    IF _runOneStep THEN
        _runOneStep := FALSE;
        RETURN;
    END_IF
END_IF

IF SUPER^.Step(1008, TRUE, 'Step number 1008') THEN
    SUPER^.StepCompleteWhen((_runOneStep OR _runAllSteps) AND _finishStep);

    IF _runOneStep THEN
        _runOneStep := FALSE;
        RETURN;
    END_IF
END_IF

IF SUPER^.Step(1009, TRUE, 'Step number 1009') THEN
    SUPER^.StepCompleteWhen((_runOneStep OR _runAllSteps) AND _finishStep);

    IF _runOneStep THEN
        _runOneStep := FALSE;
        RETURN;
    END_IF
END_IF

IF SUPER^.Step(1010, TRUE, 'Step number 1010') THEN
    SUPER^.StepCompleteWhen((_runOneStep OR _runAllSteps) AND _finishStep);

    IF _runOneStep THEN
        _runOneStep := FALSE;
        RETURN;
    END_IF
END_IF

IF SUPER^.Step(1011, TRUE, 'Step number 1011') THEN
    SUPER^.StepCompleteWhen((_runOneStep OR _runAllSteps) AND _finishStep);

    IF _runOneStep THEN
        _runOneStep := FALSE;
        RETURN;
    END_IF
END_IF

IF SUPER^.Step(1012, TRUE, 'Step number 1012') THEN
    SUPER^.StepCompleteWhen((_runOneStep OR _runAllSteps) AND _finishStep);

    IF _runOneStep THEN
        _runOneStep := FALSE;
        RETURN;
    END_IF
END_IF

IF SUPER^.Step(1013, TRUE, 'Step number 1013') THEN
    SUPER^.StepCompleteWhen((_runOneStep OR _runAllSteps) AND _finishStep);

    IF _runOneStep THEN
        _runOneStep := FALSE;
        RETURN;
    END_IF
END_IF

IF SUPER^.Step(1014, TRUE, 'Step number 1014') THEN
    SUPER^.StepCompleteWhen((_runOneStep OR _runAllSteps) AND _finishStep);

    IF _runOneStep THEN
        _runOneStep := FALSE;
        RETURN;
    END_IF
END_IF

IF SUPER^.Step(1015, TRUE, 'Step number 1015') THEN
    SUPER^.StepCompleteWhen((_runOneStep OR _runAllSteps) AND _finishStep);

    IF _runOneStep THEN
        _runOneStep := FALSE;
        RETURN;
    END_IF
END_IF

IF SUPER^.Step(1016, TRUE, 'Step number 1016') THEN
    SUPER^.StepCompleteWhen((_runOneStep OR _runAllSteps) AND _finishStep);

    IF _runOneStep THEN
        _runOneStep := FALSE;
        RETURN;
    END_IF
END_IF

IF SUPER^.Step(1017, TRUE, 'Step number 1017') THEN
    SUPER^.StepCompleteWhen((_runOneStep OR _runAllSteps) AND _finishStep);

    IF _runOneStep THEN
        _runOneStep := FALSE;
        RETURN;
    END_IF
END_IF

IF SUPER^.Step(1018, TRUE, 'Step number 1018') THEN
    SUPER^.StepCompleteWhen((_runOneStep OR _runAllSteps) AND _finishStep);

    IF _runOneStep THEN
        _runOneStep := FALSE;
        RETURN;
    END_IF
END_IF

IF SUPER^.Step(1019, TRUE, 'Step number 1019') THEN
    SUPER^.StepCompleteWhen((_runOneStep OR _runAllSteps) AND _finishStep);

    IF _runOneStep THEN
        _runOneStep := FALSE;
        RETURN;
    END_IF
END_IF

IF SUPER^.Step(1020, TRUE, 'Step number 1020') THEN
    SUPER^.StepCompleteWhen((_runOneStep OR _runAllSteps) AND _finishStep);

    IF _runOneStep THEN
        _runOneStep := FALSE;
        RETURN;
    END_IF
END_IF

IF SUPER^.Step(1021, TRUE, 'Step number 1021') THEN
    SUPER^.StepCompleteWhen((_runOneStep OR _runAllSteps) AND _finishStep);

    IF _runOneStep THEN
        _runOneStep := FALSE;
        RETURN;
    END_IF
END_IF

IF SUPER^.Step(1022, TRUE, 'Step number 1022') THEN
    SUPER^.StepCompleteWhen((_runOneStep OR _runAllSteps) AND _finishStep);

    IF _runOneStep THEN
        _runOneStep := FALSE;
        RETURN;
    END_IF
END_IF

IF SUPER^.Step(1023, TRUE, 'Step number 1023') THEN
    SUPER^.StepCompleteWhen((_runOneStep OR _runAllSteps) AND _finishStep);

    IF _runOneStep THEN
        _runOneStep := FALSE;
        RETURN;
    END_IF
END_IF

//******************************************************************
IF SUPER^.Step(_stepId, _enabled, _stepDescription) THEN
    SUPER^.StepCompleteWhen((_runOneStep OR _runAllSteps) AND _finishStep);

    IF _runOneStep THEN
        _runOneStep := FALSE;
        RETURN;
    END_IF
END_IF
END_METHOD

METHOD PROTECTED OnSequenceCompleted
_onSequenceCompleteCount := _onSequenceCompleteCount + 1;
END_METHOD

METHOD PROTECTED OnSequencerError
VAR_INPUT
    inErrorId : eSequencerError;
END_VAR
CASE inErrorId OF
    eSequencerError.noError:
        _onSequencerErrorCount := _onSequencerErrorCount + 0;
    eSequencerError.NotUniqueStepId:
        _onSequencerErrorCount := _onSequencerErrorCount + 10;
    eSequencerError.StepIdHasBeenChanged:
        _onSequencerErrorCount := _onSequencerErrorCount + 20;
    eSequencerError.OrderOfTheStepHasBeenChanged:
        _onSequencerErrorCount := _onSequencerErrorCount + 40;
    eSequencerError.StepWithRequestedIdDoesNotExists:
        _onSequencerErrorCount := _onSequencerErrorCount + 50;
    eSequencerError.MultipleRequestStepMethodCall:
        _onSequencerErrorCount := _onSequencerErrorCount + 60;
    eSequencerError.StepIdTooLow:
        _onSequencerErrorCount := _onSequencerErrorCount + 70;
    eSequencerError.StepIdTooHigh:
        _onSequencerErrorCount := _onSequencerErrorCount + 80;
ELSE
    _onSequencerErrorCount := _onSequencerErrorCount + 0;
END_CASE
END_METHOD

METHOD PROTECTED OnStateChange
VAR_INPUT
    PreviousState : INT;
    NewState : INT;
END_VAR
THIS^._onStateChangeCount := THIS^._onStateChangeCount + 1;
_stateChangeFrom := PreviousState;
_stateChangeTo := NewState;

IF _callRestoreInOnStateChange THEN
    Restore();
END_IF
END_METHOD

METHOD PROTECTED OnStepCompleted
_onCompleteStepCount := _onCompleteStepCount + 1;
END_METHOD

PROPERTY INTERNAL RequestStepCycle : UINT
GET
RequestStepCycle := _requestStepCycle;
END_GET
SET
_requestStepCycle := RequestStepCycle;
END_SET
END_PROPERTY

METHOD INTERNAL SequencerClose
SUPER^._Close();
END_METHOD

METHOD INTERNAL SequencerHasError : BOOL
SequencerHasError := SUPER^._sequencerHasError;
END_METHOD

METHOD INTERNAL SequencerOpen
SUPER^._Open();
END_METHOD

METHOD INTERNAL SetChildState
VAR_INPUT
    inState : INT;
END_VAR
THIS^._myTcoState.ChangeState(inState);
END_METHOD

METHOD INTERNAL SetCurrentStep
VAR_INPUT
    inStepID : INT;
    inStepDescription : STRING(254);
END_VAR
THIS^._currentStep.ID := inStepID;
THIS^._currentStep.Description := inStepDescription;
END_METHOD

METHOD SetCurrentStepToErrorState : BOOL
_currentStep.Status := TcoCore.eStepStatus.Error;
SetCurrentStepToErrorState := _currentStep.Status = TcoCore.eStepStatus.Error;
END_METHOD

METHOD SetCyclicMode : BOOL
ModeController.Mode := eSequencerMode.CyclicMode;
SetCyclicMode := ModeController.Mode = eSequencerMode.CyclicMode;
END_METHOD

METHOD SetInvalidMode : BOOL
ModeController.Mode := eSequencerMode.Invalid;
SetInvalidMode := ModeController.Mode = eSequencerMode.Invalid;
END_METHOD

METHOD INTERNAL SetNumberOfSteps
VAR_INPUT
    inNumberOfSteps : UINT;
END_VAR
_stepCounter := inNumberOfSteps;
_numberOfStepsInSequence := inNumberOfSteps;
_previousNumberOfStepsInSequence := inNumberOfSteps;
END_METHOD

METHOD INTERNAL SetSequenceAsChecked
_stepIDUniquenessChecked := TRUE;
_StepIdUniquenessControlState := eStepIdUniquenessControlState.Done;
END_METHOD

METHOD INTERNAL SetSequenceAsNotChecked
_stepIDUniquenessChecked := FALSE;
_StepIdUniquenessControlState := eStepIdUniquenessControlState.NotYetStarted;
END_METHOD

METHOD SetStepMode : BOOL
ModeController.Mode := eSequencerMode.StepMode;
SetStepMode := ModeController.Mode = eSequencerMode.StepMode;
END_METHOD

METHOD INTERNAL SetTestParams
VAR_INPUT
    inRunOneStep : BOOL;
    inRunAllSteps : BOOL;
    inFinishStep : BOOL;
    inID : UINT;
    inEnabled : BOOL;
    inStepDescription : STRING(254);
END_VAR
THIS^._runOneStep := inRunOneStep;
THIS^._runAllSteps := inRunAllSteps;
THIS^._finishStep := inFinishStep;
THIS^._stepId := inID;
THIS^._enabled := inEnabled;
THIS^._stepDescription := inStepDescription;
END_METHOD

METHOD StepCount
VAR_INPUT
    inTotalStepNumber : UINT;
    inFinishStep : BOOL;
END_VAR
VAR
    i : INT;
    _lastStepId : INT;
END_VAR
FOR i := 0 TO inTotalStepNumber DO
    IF SUPER^.Step(i, TRUE, CONCAT('Step number ', INT_TO_STRING(i))) THEN
        SUPER^.StepCompleteWhen(inFinishStep);
    END_IF
END_FOR
END_METHOD

{attribute 'TcRpcEnable'}
METHOD INTERNAL UpdateCurrentStepDetails
_currentStepId := SUPER^._currentStep.ID;
_currentStepOrder := SUPER^._currentStep.Order;
_currentStepEnabled := SUPER^._currentStep.Enabled;
_currentStepDescription := SUPER^._currentStep.Description;
_currentStepStatus := SUPER^._currentStep.Status;
_currentStepDuration := SUPER^._currentStep.Duration;
END_METHOD

END_FUNCTION_BLOCK

// ---- Tests/TcoSequence/TcoSequenceNonAutoRestorableTest.TcPOU
FUNCTION_BLOCK TcoSequenceNonAutoRestorableTest EXTENDS TcoCore._internals_TcoContext
VAR
    _callMyPlcInstance : BOOL := FALSE;
    _sequencer : _TcoSequence(THIS^, eRestoreMode.None);
    _runPLCinstanceOnce : BOOL := FALSE;
    _runPLCinstanceCyclicaly : BOOL := FALSE;
    _stepID : INT := 32764;
    _enabled : BOOL;
    _stepDescription : STRING := 'Last step sequence message';
    _runOneStep : BOOL;
    _runAllSteps : BOOL;
    _finishStep : BOOL;
    _restore : BOOL;
    _cycleCount : INT;
    _restoreCycleCount : INT;
    _init : BOOL;
END_VAR

IF _callMyPlcInstance THEN
    IF NOT _init THEN
        ContextOpen();
        ContextClose();
        _init := THIS^._rtc.IsValid;
    END_IF

    IF _restore THEN
        ContextOpen();
        THIS^._sequencer.Restore();
        _restoreCycleCount := _restoreCycleCount + 1;
        _restore := FALSE;
        ContextClose();
        RETURN;
    END_IF

    IF _runPLCinstanceOnce AND NOT _runPLCinstanceCyclicaly THEN
        ContextOpen();
        THIS^.PLCinstanceRun(_stepID, _enabled, _stepDescription);
        _cycleCount := _cycleCount + 1;
        _runPLCinstanceOnce := FALSE;
        ContextClose();
    END_IF

    IF _runPLCinstanceCyclicaly AND NOT _runPLCinstanceOnce THEN
        ContextOpen();
        THIS^.PLCinstanceRun(_stepID, _enabled, _stepDescription);
        _cycleCount := _cycleCount + 1;
        ContextClose();
    END_IF
END_IF;

{attribute 'TcRpcEnable'}
METHOD ChildHasAutoRestoreEnabled : BOOL;
ChildHasAutoRestoreEnabled := _sequencer.ChildHasAutoRestoreEnabled();
END_METHOD

{attribute 'TcRpcEnable'}
METHOD ChildIsAutoRestorable : BOOL;
ChildIsAutoRestorable := _sequencer.ChildIsAutoRestorable();
END_METHOD

{attribute 'TcRpcEnable'}
METHOD CleanupPointers
_sequencer.CleanupPointers();
END_METHOD

{attribute 'TcRpcEnable'}
METHOD ClearNumberOfSteps
_sequencer.ClearNumberOfSteps();
END_METHOD

{attribute 'TcRpcEnable'}
METHOD PROTECTED ContextClose
SUPER^._Close();
END_METHOD

{attribute 'TcRpcEnable'}
METHOD ContextOpen
SUPER^._Open();
END_METHOD

{attribute 'TcRpcEnable'}
METHOD GetChildState : INT
GetChildState := _sequencer.GetChildState();
END_METHOD

{attribute 'TcRpcEnable'}
METHOD GetCurrentStepOrder : UINT
GetCurrentStepOrder := _sequencer._currentStep.Order;
END_METHOD

{attribute 'TcRpcEnable'}
METHOD GetNumberOfStepsInSequence : UINT
GetNumberOfStepsInSequence := _sequencer._numberOfStepsInSequence;
END_METHOD

{attribute 'TcRpcEnable'}
METHOD GetOrderOfTheCurrentlyEvaluatedStep : UINT
GetOrderOfTheCurrentlyEvaluatedStep := _sequencer._theOrderOfTheCurrentlyEvaluatedStep;
END_METHOD

{attribute 'TcRpcEnable'}
METHOD GetOrderOfTheCurrentlyExecutedStep : UINT
GetOrderOfTheCurrentlyExecutedStep := _sequencer._theOrderOfTheCurrentlyExecutedStep;
END_METHOD

{attribute 'TcRpcEnable'}
METHOD GetPreviousNumberOfStepsInSequence : UINT
GetPreviousNumberOfStepsInSequence := _sequencer._previousNumberOfStepsInSequence;
END_METHOD

{attribute 'TcRpcEnable'}
METHOD GetRequestStepCycle : UINT
GetRequestStepCycle := _sequencer.RequestStepCycle;
END_METHOD

{attribute 'TcRpcEnable'}
METHOD GetSequencerErrorId : INT
GetSequencerErrorId := _sequencer.GetSequencerErrorId();
END_METHOD

{attribute 'TcRpcEnable'}
METHOD GetTextOfTheMostImportantMessage : STRING(254)
GetTextOfTheMostImportantMessage := THIS^._sequencer.GetTextOfTheMostImportantMessage();
END_METHOD

{attribute 'TcRpcEnable'}
METHOD HasAutoRestoreEnabled : BOOL;
HasAutoRestoreEnabled := _sequencer.HasAutoRestoreEnabled();
END_METHOD

{attribute 'TcRpcEnable'}
METHOD IsAutoRestorable : BOOL;
IsAutoRestorable := _sequencer.IsAutoRestorable();
END_METHOD

{attribute 'TcRpcEnable'}
METHOD IsFirstStepEntry : BOOL
IsFirstStepEntry := THIS^._sequencer.IsFirstStepEntry();
END_METHOD

METHOD PROTECTED Main
END_METHOD

{attribute 'TcRpcEnable'}
METHOD PLCinstanceRun
VAR_INPUT
    inStepId : UINT;
    inEnabled : BOOL;
    inStepDescription : STRING(254);
END_VAR
THIS^._sequencer.SetTestParams(_runOneStep,
    _runAllSteps,
    _finishStep,
    inStepId,
    inEnabled,
    inStepDescription);

THIS^._sequencer._RunExecutionSubstitute();
END_METHOD

{attribute 'TcRpcEnable'}
METHOD RequestStep
VAR_INPUT
    inRequestedStepId : INT;
END_VAR
_sequencer._RequestStep(inRequestedStepId);
END_METHOD

{attribute 'TcRpcEnable'}
METHOD Restore
_sequencer.Restore();
END_METHOD

{attribute 'TcRpcEnable'}
METHOD SequenceComplete
_sequencer._SequenceComplete();
END_METHOD

{attribute 'TcRpcEnable'}
METHOD SequencerClose
THIS^._sequencer.SequencerClose();
END_METHOD

{attribute 'TcRpcEnable'}
METHOD SequencerHasError : BOOL
SequencerHasError := _sequencer.SequencerHasError();
END_METHOD

{attribute 'TcRpcEnable'}
METHOD SequencerOpen
THIS^._sequencer.SequencerOpen();
END_METHOD

{attribute 'TcRpcEnable'}
METHOD SetChildState
VAR_INPUT
    inState : INT;
END_VAR
_sequencer.SetChildState(inState);
END_METHOD

{attribute 'TcRpcEnable'}
METHOD SetCurrentStep
VAR_INPUT
    inStepID : INT;
    inStepDescription : STRING(254);
END_VAR
_sequencer.SetCurrentStep(inStepID := inStepID, inStepDescription := inStepDescription);
END_METHOD

{attribute 'TcRpcEnable'}
METHOD SetCurrentStepToErrorState : BOOL
SetCurrentStepToErrorState := _sequencer.SetCurrentStepToErrorState();
END_METHOD

{attribute 'TcRpcEnable'}
METHOD SetCyclicMode : BOOL
SetCyclicMode := _sequencer.SetCyclicMode();
END_METHOD

{attribute 'TcRpcEnable'}
METHOD SetInvalidMode : BOOL
SetInvalidMode := _sequencer.SetInvalidMode();
END_METHOD

{attribute 'TcRpcEnable'}
METHOD SetNumberOfSteps : UINT
VAR_INPUT
    inNumberOfSteps : UINT;
END_VAR
_sequencer.SetNumberOfSteps(inNumberOfSteps);
SetNumberOfSteps := _sequencer._numberOfStepsInSequence;
END_METHOD

{attribute 'TcRpcEnable'}
METHOD SetRequestStepCycle : UINT
VAR_INPUT
    Value : UINT;
END_VAR
_sequencer.RequestStepCycle := Value;
SetRequestStepCycle := _sequencer.RequestStepCycle;
END_METHOD

{attribute 'TcRpcEnable'}
METHOD SetSequenceAsChecked : BOOL
VAR_INPUT
END_VAR
_sequencer.SetSequenceAsChecked();
END_METHOD

{attribute 'TcRpcEnable'}
METHOD SetSequenceAsNotChecked : BOOL
VAR_INPUT
END_VAR
_sequencer.SetSequenceAsNotChecked();
END_METHOD

{attribute 'TcRpcEnable'}
METHOD SetStepMode : BOOL
SetStepMode := _sequencer.SetStepMode();
END_METHOD

{attribute 'TcRpcEnable'}
METHOD Step : BOOL
VAR_INPUT
    inStepId : INT;
    inEnabled : BOOL;
    inStepDescription : STRING(254);
END_VAR
Step := _sequencer._Step(inStepID := inStepId, inEnabled := inEnabled, inStepDescription := inStepDescription);
END_METHOD

{attribute 'TcRpcEnable'}
METHOD StepBackward
_sequencer._StepBackward();
END_METHOD

{attribute 'TcRpcEnable'}
METHOD StepCompleteWhen
VAR_INPUT
    inCondition : BOOL;
END_VAR
_sequencer._StepCompleteWhen(inCondition);
END_METHOD

{attribute 'TcRpcEnable'}
METHOD StepForward
_sequencer._StepForward();
END_METHOD

{attribute 'TcRpcEnable'}
METHOD StepIn
_sequencer._StepIn();
END_METHOD

{attribute 'TcRpcEnable'}
METHOD UpdateCurrentStepDetails
VAR_INPUT
END_VAR
_sequencer.UpdateCurrentStepDetails();
END_METHOD

END_FUNCTION_BLOCK

// ---- Tests/TcoMessenger/TcoMessengerContextTest.TcPOU
FUNCTION_BLOCK TcoMessengerContextTest EXTENDS TcoCore._internals_TcoContext
VAR
    _callMyPlcInstanceRtcUpdate : BOOL := FALSE;
    _callMyPlcInstanceRun : BOOL := FALSE;
    _nowLocal : DATE_AND_TIME;
    _nowUtc : DATE_AND_TIME;
    _rtcIsValid : BOOL := FALSE;
    _rtcIsSynchronized : BOOL := FALSE;
    {attribute addProperty Name "this is the name of messenger test"}
    _tcoMessangerTests : TcoMessengerTests(THIS^);
END_VAR

IF THIS^._callMyPlcInstanceRtcUpdate THEN
    THIS^._rtcUpdate();
    _nowLocal := THIS^.RealTimeClock.NowLocal();
    _nowUtc := THIS^.RealTimeClock.NowUTC();
    _rtcIsValid := THIS^.RealTimeClock.IsValid;
    _rtcIsSynchronized := THIS^.RealTimeClock.IsSynchronized;
END_IF

IF THIS^._callMyPlcInstanceRun THEN
    THIS^.Run();
END_IF

{attribute 'TcRpcEnable'}
METHOD INTERNAL ContextClose
SUPER^._Close();
END_METHOD

{attribute 'TcRpcEnable'}
METHOD INTERNAL ContextOpen
SUPER^._Open();
END_METHOD

METHOD PROTECTED Main
END_METHOD

{attribute 'TcRpcEnable'}
METHOD INTERNAL RtcIsValid : BOOL
RtcIsValid := THIS^.RealTimeClock.IsValid;
_rtcIsValid := THIS^.RealTimeClock.IsValid;
END_METHOD

END_FUNCTION_BLOCK

// ---- Tests/TcoMessenger/TcoMessengerTests.TcPOU
FUNCTION_BLOCK TcoMessengerTests EXTENDS TcoCore.TcoObject
VAR
    _category : TcoCore.eMessageCategory;
    _minLevel : TcoCore.eMessageCategory;
    _messageDigestMethod : TcoCore.eMessageDigestMethod;
    _messageLoggingMethod : TcoCore.eMessengerLogMethod;
END_VAR
VAR
    _BOOL : BOOL := TRUE;
    _BYTE : BYTE := 1;
    _WORD : WORD := 22;
    _DWORD : DWORD := 333;
    _LWORD : LWORD := 4444;
    _SINT : SINT := 12;
    _USINT : USINT := 13;
    _INT : INT := 14;
    _UINT : UINT := 55;
    _DINT : DINT := 66;
    _UDINT : UDINT := 77;
    _LINT : LINT := 88;
    _ULINT : ULINT := 99;
    _LTIME : LTIME := LTIME#551US615NS;
    _Real : REAL := 99.9;
    _LReal : LREAL := 88.8;
    _DateAndTime : DATE_AND_TIME := DT#2106-02-06-06:28:15;
    _Date : DATE := D#2106-02-06;
    _Time : TIME := T#71582M47S295MS;
    _WString : WSTRING := "W1";
    _TOD : TOD := TOD#23:59:59.999;
    _String : STRING := 'S1';
END_VAR

{attribute 'TcRpcEnable'}
METHOD AppendAnys_1 : BOOL
VAR_INPUT
END_VAR
_messenger.Build()
    .AppendAny(_BOOL)
    .AppendAny(_BYTE)
    .AppendAny(_WORD)
    .AppendAny(_DWORD)
    .AppendAny(_LWORD)
    .AppendAny(_SINT)
    .AppendAny(_USINT)
    .AppendAny(_INT)
    .AppendAny(_UINT)
    .AppendAny(_DINT)
    .AppendAny(_UDINT)
    .As().AsDebug();
END_METHOD

{attribute 'TcRpcEnable'}
METHOD AppendAnys_2 : BOOL
VAR_INPUT
END_VAR
_messenger.Build()
    .AppendAny(_LINT)
    .AppendAny(_ULINT)
    .AppendAny(_LTIME)
    .AppendAny(_Real)
    .AppendAny(_LReal)
    .AppendAny(_DateAndTime)
    .AppendAny(_Date)
    .AppendAny(_Time)
    .AppendAny(_WString)
    .AppendAny(_TOD)
    .AppendAny(_String)
    .As().AsDebug();
END_METHOD

{attribute 'TcRpcEnable'}
METHOD AsDebug : BOOL
VAR_INPUT
    TextMessage1 : STRING;
    TextMessage2 : STRING;
    Value : LREAL;
END_VAR
_messenger.Build().Append(TextMessage1).Append(TextMessage2).AppendAny(Value).As().AsDebug();
END_METHOD

{attribute 'TcRpcEnable'}
METHOD AsError : BOOL
VAR_INPUT
    TextMessage1 : STRING;
    TextMessage2 : STRING;
    Value : LREAL;
END_VAR
_messenger.Build().Append(TextMessage1).Append(TextMessage2).AppendAny(Value).As().AsError();
END_METHOD

{attribute 'TcRpcEnable'}
METHOD AsFatal : BOOL
VAR_INPUT
    TextMessage1 : STRING;
    TextMessage2 : STRING;
    Value : LREAL;
END_VAR
_messenger.Build().Append(TextMessage1).Append(TextMessage2).AppendAny(Value).As().AsFatal();
END_METHOD

{attribute 'TcRpcEnable'}
METHOD AsInfo : BOOL
VAR_INPUT
    TextMessage1 : STRING;
    TextMessage2 : STRING;
    Value : LREAL;
END_VAR
_messenger.Build().Append(TextMessage1).Append(TextMessage2).AppendAny(Value).As().AsInfo();
END_METHOD

{attribute 'TcRpcEnable'}
METHOD AsTrace : BOOL
VAR_INPUT
    TextMessage1 : STRING;
    TextMessage2 : STRING;
    Value : LREAL;
END_VAR
_messenger.Build().Append(TextMessage1).Append(TextMessage2).AppendAny(Value).As().AsTrace();
END_METHOD

{attribute 'TcRpcEnable'}
METHOD AsWarning : BOOL
VAR_INPUT
    TextMessage1 : STRING;
    TextMessage2 : STRING;
    Value : LREAL;
END_VAR
_messenger.Build().Append(TextMessage1).Append(TextMessage2).AppendAny(Value).As().AsWarning();
END_METHOD

{attribute 'TcRpcEnable'}
METHOD INTERNAL Catastrophic
VAR_INPUT
    Message : STRING(255);
END_VAR
_messenger.Catastrophic(Message);
END_METHOD

{attribute 'TcRpcEnable'}
METHOD INTERNAL Critical
VAR_INPUT
    Message : STRING(255);
END_VAR
_messenger.Critical(Message);
END_METHOD

{attribute 'TcRpcEnable'}
METHOD INTERNAL Debug
VAR_INPUT
    Message : STRING(255);
END_VAR
_messenger.Debug(Message);
END_METHOD

{attribute 'TcRpcEnable'}
METHOD INTERNAL Error
VAR_INPUT
    Message : STRING(255);
END_VAR
_messenger.Error(Message);
END_METHOD

{attribute 'TcRpcEnable'}
METHOD INTERNAL Info
VAR_INPUT
    Message : STRING(255);
END_VAR
_messenger.Info(Message);
END_METHOD

{attribute 'TcRpcEnable'}
METHOD INTERNAL Notify
VAR_INPUT
    Message : STRING(255);
END_VAR
_messenger.Notify(Message);
END_METHOD

{attribute 'TcRpcEnable'}
METHOD OnCondition : BOOL
VAR_INPUT
    inCondition : BOOL;
    message : STRING;
END_VAR
_messenger.OnCondition(inCondition).Post(message, _category);
END_METHOD

{attribute 'TcRpcEnable'}
METHOD Pin : BOOL
VAR_INPUT
    inCondition : BOOL;
    message : STRING;
END_VAR
IF (inCondition) THEN
    _messenger.Post(message, _category).Pin();
ELSE
    _messenger.Post(message, _category);
END_IF;
END_METHOD

{attribute 'TcRpcEnable'}
METHOD Pinned : BOOL
Pinned := _messenger.Pinned;
END_METHOD

{attribute 'TcRpcEnable'}
METHOD INTERNAL Post
VAR_INPUT
    Message : STRING(255);
END_VAR
_messenger.Post(Message, _category);
END_METHOD

{attribute 'TcRpcEnable'}
METHOD INTERNAL Programming
VAR_INPUT
    Message : STRING(255);
END_VAR
_messenger.Programming(Message);
END_METHOD

{attribute 'TcRpcEnable'}
METHOD INTERNAL Resume
Context.Environment.Messaging.Resume();
END_METHOD

{attribute 'TcRpcEnable'}
METHOD INTERNAL SetMessageDigestMethod
Context.Environment.Messaging.MessageDigestMethod := _messageDigestMethod;
END_METHOD

{attribute 'TcRpcEnable'}
METHOD INTERNAL SetMessageLoggingMethod
Context.Environment.Messaging.MessengerLoggingMethod := _messageLoggingMethod;
END_METHOD

{attribute 'TcRpcEnable'}
METHOD INTERNAL SetMinLevel
Context.Environment.Messaging.MinLevel := _minLevel;
END_METHOD

{attribute 'TcRpcEnable'}
METHOD INTERNAL Suspend
Context.Environment.Messaging.Suspend();
END_METHOD

{attribute 'TcRpcEnable'}
METHOD INTERNAL TimedOut
VAR_INPUT
    Message : STRING(255);
END_VAR
_messenger.Warning(Message);
END_METHOD

{attribute 'TcRpcEnable'}
METHOD INTERNAL Trace
VAR_INPUT
    Message : STRING(255);
END_VAR
_messenger.Trace(Message);
END_METHOD

{attribute 'TcRpcEnable'}
METHOD UnPin : BOOL
VAR_INPUT
    inCondition : BOOL;
    message : STRING;
END_VAR
_messenger.UnPin();
END_METHOD

{attribute 'TcRpcEnable'}
METHOD INTERNAL Warning
VAR_INPUT
    Message : STRING(255);
END_VAR
_messenger.Warning(Message);
END_METHOD

END_FUNCTION_BLOCK

// ---- Tests/TcoMessenger/TcoContextMessagingPerf.TcPOU
FUNCTION_BLOCK TcoContextMessagingPerf EXTENDS TcoContextTest
VAR
    _lot_of_messages : ARRAY[0.._messagesUpperBound] OF TcoCore.TcoMessenger(THIS^);
    _numberOfTestMessages : INT;
END_VAR
VAR CONSTANT
    _messagesUpperBound : INT := 10000;
END_VAR

METHOD PROTECTED Main
VAR
    index : INT;
END_VAR
IF (_numberOfTestMessages > _messagesUpperBound) THEN
    _numberOfTestMessages := _messagesUpperBound;
END_IF

FOR index := 0 TO _numberOfTestMessages DO
    THIS^._lot_of_messages[index].Info(INT_TO_STRING(index));
END_FOR
END_METHOD

END_FUNCTION_BLOCK

// ---- Tests/TcoComponent/TcoComponentTest.TcPOU
FUNCTION_BLOCK TcoComponentTest EXTENDS TcoCore._internals_TcoContext
VAR
    _callMyPlcInstance : BOOL := FALSE;
    _component : _TcoComponent(THIS^);
    _runPLCinstanceOnce : BOOL := FALSE;
    _runPLCinstanceCyclicaly : BOOL := FALSE;
    _restore : BOOL;
    _cycleCount : INT;
    _restoreCycleCount : INT;
    _init : BOOL;
END_VAR

IF _callMyPlcInstance THEN
    IF NOT _init THEN
        ContextOpen();
        ContextClose();
        _init := THIS^._rtc.IsValid;
    END_IF

    IF _restore THEN
        ContextOpen();
        THIS^._component.Restore();
        _restoreCycleCount := _restoreCycleCount + 1;
        _restore := FALSE;
        ContextClose();
        RETURN;
    END_IF

    IF _runPLCinstanceOnce AND NOT _runPLCinstanceCyclicaly THEN
        ContextOpen();
        THIS^.PLCinstanceRun();
        _cycleCount := _cycleCount + 1;
        _runPLCinstanceOnce := FALSE;
        ContextClose();
    END_IF

    IF _runPLCinstanceCyclicaly AND NOT _runPLCinstanceOnce THEN
        ContextOpen();
        THIS^.PLCinstanceRun();
        _cycleCount := _cycleCount + 1;
        ContextClose();
    END_IF
END_IF;

{attribute 'TcRpcEnable'}
METHOD INTERNAL ContextClose
SUPER^._Close();
END_METHOD

{attribute 'TcRpcEnable'}
METHOD INTERNAL ContextOpen
SUPER^._Open();
END_METHOD

{attribute 'TcRpcEnable'}
METHOD INTERNAL IsService : BOOL
IsService := THIS^._component.IsService;
END_METHOD

METHOD PROTECTED Main
END_METHOD

{attribute 'TcRpcEnable'}
METHOD INTERNAL PLCinstanceRun
THIS^._component();
END_METHOD

METHOD PROTECTED Restore
THIS^._component.Restore();
END_METHOD

{attribute 'TcRpcEnable'}
METHOD INTERNAL Service
THIS^._component.Service();
END_METHOD

{attribute 'TcRpcEnable'}
METHOD INTERNAL TriggerRestore
THIS^.Restore();
END_METHOD

END_FUNCTION_BLOCK

// ---- Tests/TcoComponent/_TcoComponent.TcPOU
FUNCTION_BLOCK _TcoComponent EXTENDS TcoCore.TcoComponent
VAR
    _task : TcoTaskTest(THIS^);
    _serviceModeCount : ULINT;
END_VAR

_task();

{attribute 'TcRpcEnable'}
METHOD INTERNAL CallBodyFromTest
_task();
END_METHOD

(*~
    <docu>
        <summary>
            Restores this instance to the Ready state. Can be called explicitly or from within one of the restore mechanisms.
        </summary>
    </docu>
~*)
METHOD Restore : ITcoRestorable
_task.Restore();
END_METHOD

METHOD PROTECTED ServiceMode
_serviceModeCount := _serviceModeCount + 1;
END_METHOD

END_FUNCTION_BLOCK

// ---- Tests/Utilities/StringBuilderTests.TcPOU
FUNCTION_BLOCK StringBuilderTests
VAR
    StringBuilder : TcoCore.StringBuilder();
    StringBuilderResult : STRING;
END_VAR

{attribute 'TcRpcEnable'}
METHOD Append
VAR_INPUT
    ToAppend : STRING;
END_VAR
StringBuilder.Append(ToAppend);
StringBuilderResult := StringBuilder._workString;
END_METHOD

{attribute 'TcRpcEnable'}
METHOD AppendAnyTest
StringBuilder.Clear();
// There was a strange compile-time error here... about function requiring exactly one input... could not get arround that... next time...
// 'AppendAny' is internal in the production code
//				     .AppendAny(_bool);
//					 .AppendAny(_real)
//					 .AppendAny(_lreal)
//					 .AppendAny(_dt)
//					 .AppendAny(_d)
//					 .AppendAny(_time)
//					 .AppendAny(_string)
//					 .AppendAny(_wstring)
//					 .AppendAny(_tod)
//					 .AppendAny(_int);
StringBuilderResult := StringBuilder._workString;
END_METHOD

{attribute 'TcRpcEnable'}
METHOD Clear
StringBuilder.Clear();
StringBuilderResult := StringBuilder._workString;
END_METHOD

{attribute 'TcRpcEnable'}
METHOD FluentApi : STRING
FluentApi :=
    StringBuilder.Clear().Append('1').Append('2').Append('3').Append('4').Clear().Append('1').Append('2').Append('3').Append('4').ToString();
END_METHOD

{attribute 'TcRpcEnable'}
METHOD ToString : STRING
ToString := StringBuilder.ToString();
StringBuilderResult := StringBuilder._workString;
END_METHOD

END_FUNCTION_BLOCK

// ---- Tests/TcoTask/PlcExecuted/TcoTaskTestContext.TcPOU
FUNCTION_BLOCK TcoTaskTestContext EXTENDS TcoCore._internals_TcoContext
VAR
    _sut : TcoCore.TcoTask(THIS^);
    _to_A : TcoTaskPlcTestObject(THIS^);
    _to_B : TcoTaskPlcTestObject(THIS^);
    _elapsedTimeETA : TIME;
    _elapsedTime : TIME;
    _runElapsedTimer : BOOL;
    _elapsedTimeTimer : Tc2_Standard.TON;
    _inBool : BOOL;
    _inUint : UINT;
    _inString : STRING;
    _retBool : BOOL;
    _retUint : UINT;
    _retString : STRING;
    _done : BOOL;
    _arranged : BOOL;
    _startCycles : ULINT;
    _endCycles : ULINT;
    _myIdentity : ULINT;
END_VAR

{attribute 'TcRpcEnable'}
METHOD _ClearPlcCycleCounter
ClearPlcCycleCounter();
END_METHOD

METHOD PROTECTED Main
_elapsedTimeTimer(IN := _runElapsedTimer, PT := _elapsedTimeETA);

CASE _testId OF
    {region "CallTasksBodiesOnly"}
    eTcoTaskTests.CallTasksBodiesOnly:
        _to_A();
        {endregion}
        {region "RestoreTasks"}
    eTcoTaskTests.RestoreTasks:
        _to_A._sut_A.Restore();
        _to_A._sut_B.Restore();
        _to_A();
        {endregion}
        {region "T300_TaskInvokeAndWaitForDone"}
    eTcoTaskTests.TaskInvokeAndWaitForDone:
        IF NOT _arranged THEN
            _to_A._sut_A.Restore();
            _to_A._sut_B.Restore();
            _to_A._sut_A.SetPreviousStateToReady();
            _to_A._sut_B.SetPreviousStateToReady();
            _arranged := TRUE;
        END_IF

        IF NOT _done THEN
            _to_A._sut_A.Invoke();
            _to_A._sut_B.Invoke();
            _to_A();
            _done := _to_A._sut_A.Done AND _to_A._sut_B.Done;
        END_IF

        IF _done THEN
            _to_A._sut_A.ReadOutState();
            _to_A._sut_B.ReadOutState();
            ProbeDoneWhen(_done);
        END_IF
        {endregion}
        {region "T301_TaskInvokeAfterDoneWithNoEmptyCycles"}
    eTcoTaskTests.TaskInvokeAfterDoneWithNoEmptyCycles:
        IF NOT _done THEN
            _to_A._sut_A.Invoke();
            _to_A._sut_B.Invoke();
            _to_A();
            _done := _to_A._sut_A.Done AND _to_A._sut_B.Done;
        END_IF

        IF _done THEN
            _to_A._sut_A.ReadOutState();
            _to_A._sut_B.ReadOutState();
            ProbeDoneWhen(_done);
        END_IF
        {endregion}
        {region "T302_TaskInvokeAfterDoneWithOneEmptyCycle"}
    eTcoTaskTests.TaskInvokeAfterDoneWithOneEmptyCycle:
        IF NOT _arranged THEN
            _arranged := TRUE;
            _plcCycleCounter := 0;
            RETURN;
        END_IF

        IF NOT _done THEN
            _to_A._sut_A.Invoke();
            _to_A._sut_B.Invoke();
            _to_A();
            _done := _to_A._sut_A.Done AND _to_A._sut_B.Done;
        END_IF

        IF _done THEN
            _to_A._sut_A.ReadOutState();
            _to_A._sut_B.ReadOutState();
            ProbeDoneWhen(_done);
        END_IF
        {endregion}
        {region "T303_TaskInvokeAfterDoneWithAbortCall"}
    eTcoTaskTests.TaskInvokeAfterDoneWithAbortCall:
        IF NOT _arranged THEN
            _to_A._sut_A.Abort();
            _to_A._sut_B.Abort();
            _arranged := TRUE;
        END_IF

        IF NOT _done THEN
            _to_A._sut_A.Invoke();
            _to_A._sut_B.Invoke();
            _to_A();
            _done := _to_A._sut_A.Done AND _to_A._sut_B.Done;
        END_IF

        IF _done THEN
            _to_A._sut_A.ReadOutState();
            _to_A._sut_B.ReadOutState();
            ProbeDoneWhen(_done);
        END_IF
        {endregion}
        {region "T304_TaskInvokeAfterDoneWithRestoreCall"}
    eTcoTaskTests.TaskInvokeAfterDoneWithRestoreCall:
        IF NOT _arranged THEN
            _to_A._sut_A.Restore();
            _to_A._sut_B.Restore();
            _arranged := TRUE;
        END_IF

        IF NOT _done THEN
            _to_A._sut_A.Invoke();
            _to_A._sut_B.Invoke();
            _to_A();
            _done := _to_A._sut_A.Done AND _to_A._sut_B.Done;
        END_IF

        IF _done THEN
            _to_A._sut_A.ReadOutState();
            _to_A._sut_B.ReadOutState();
            ProbeDoneWhen(_done);
        END_IF
        {endregion}
        {region "T305_TaskAbortDuringExecutionAndInvoke"}
    eTcoTaskTests.TaskAbortDuringExecutionAndInvoke:
        IF NOT _arranged THEN
            _arranged := TRUE;
            _plcCycleCounter := 0;
            _retBool := FALSE;
            RETURN;
        END_IF

        IF NOT _done THEN
            _to_A._sut_A.Invoke();
            _to_A._sut_B.Invoke();
            _to_A();

            IF _to_A._sut_A.Done AND NOT _retBool THEN
                _to_A._sut_A.Abort();
                _to_A._sut_B.Abort();
                _retBool := true;
            END_IF

            _done := _to_A._sut_A.Done AND _to_A._sut_B.Done;
        END_IF

        IF _done THEN
            _to_A._sut_A.ReadOutState();
            _to_A._sut_B.ReadOutState();
            ProbeDoneWhen(_done);
        END_IF
        {endregion}
        {region "T310_TaskError"}
    eTcoTaskTests.TaskError:
        IF NOT _arranged THEN
            IF _plcCycleCounter = 1 THEN
                _to_A.CounterValue_A := _inUint;
                RETURN;
            END_IF

            IF _plcCycleCounter = 2 THEN
                _to_A._sut_A.Invoke();
                RETURN;
            END_IF

            IF _plcCycleCounter > 2 AND _plcCycleCounter <= 5 THEN
                _to_A._sut_A();
                RETURN;
            END_IF

            IF _plcCycleCounter = 6 THEN
                _to_A._sut_A();
                _to_A._sut_A.ReadOutState();
                _arranged := TRUE;
                RETURN;
            END_IF
        END_IF

        IF NOT _done THEN
            IF _plcCycleCounter = 7 THEN
                _to_A.CounterValue_A := _to_A.CounterValue_A + 5;
                _to_A._sut_A();
                _to_A._sut_A.ReadOutState();
            END_IF

            IF _plcCycleCounter > 7 AND _plcCycleCounter <= 7 + _inUint THEN
                _to_A._sut_A();
                _to_A._sut_A.ReadOutState();
            END_IF

            _done := _plcCycleCounter >= 7 + _inUint;
            ProbeDoneWhen(_done);
        END_IF
        {endregion}
        {region "T311_TaskInvokeAfterErrorNoRestoreNoEmptyCycles"}
    eTcoTaskTests.TaskInvokeAfterErrorNoRestoreNoEmptyCycles:
        IF NOT _arranged THEN
            _to_A._sut_A.Invoke();
            _arranged := TRUE;
            RETURN;
        END_IF

        IF NOT _done THEN
            _to_A._sut_A();
            _to_A._sut_A.ReadOutState();
            ProbeDoneWhen(_plcCycleCounter >= 1 + _inUint);
        END_IF
        {endregion}
        {region "T312_TaskInvokeAfterErrorNoRestoreOneEmptyCycle"}
    eTcoTaskTests.TaskInvokeAfterErrorNoRestoreOneEmptyCycle:
        IF NOT _arranged THEN
            IF _plcCycleCounter = 1 THEN
                RETURN;
            END_IF

            IF _plcCycleCounter = 2 THEN
                _to_A._sut_A.Invoke();
                RETURN;
            END_IF
        END_IF

        IF NOT _done THEN
            _to_A._sut_A();
            _to_A._sut_A.ReadOutState();
            _done := _plcCycleCounter >= 2 + _inUint;
            ProbeDoneWhen(_done);
        END_IF
        {endregion}
        {region "T313_TaskInvokeAfterErrorWithRestore"}
    eTcoTaskTests.TaskInvokeAfterErrorWithRestore:
        _to_A._sut_A.Restore();
        _to_A._sut_A.Invoke();
        _to_A._sut_A();
        _to_A._sut_A.ReadOutState();
        _done := TRUE;
        ProbeDoneWhen(_done);
        {endregion}
        {region "T314_TaskAbortDuringExecution"}
    eTcoTaskTests.TaskAbortDuringExecution:
        IF _plcCycleCounter = 1 THEN
            _to_A._sut_A.Restore();
            RETURN;
        END_IF

        IF _plcCycleCounter = 2 THEN
            _to_A._sut_A.Invoke();
            _to_A._sut_A();
            _to_A._sut_A.ReadOutState();
            RETURN;
        END_IF

        IF _plcCycleCounter = 3 THEN
            _to_A._sut_A.Abort();
            _to_A._sut_A();
            _to_A._sut_A.ReadOutState();
            _done := TRUE;
            ProbeDoneWhen(_done);
        END_IF
        {endregion}
        {region "T315_TaskMessage"}
    eTcoTaskTests.TaskMessage:
        _to_A._sut_A.PostMessage(Message := _inString);
        _retString := _to_A._sut_A.GetMessage();
        _done := TRUE;
        ProbeDoneWhen(_done);
        {endregion}
        {region "T316_IdentitiesTest"}
    eTcoTaskTests.IdentitiesTest:
        _runElapsedTimer := TRUE;
        _elapsedTimeETA := UINT_TO_TIME(_inUint);
        _to_A._sut_A.ReadOutIdentities();
        _to_A.ReadOutIdentities();
        ReadOutCycleCounters();
        _done := _elapsedTimeTimer.Q;
        ProbeDoneWhen(_done);
        {endregion}
        {region "T317_CheckAutoRestoreProperties"}
    eTcoTaskTests.CheckAutoRestoreProperties:
        _to_A._tSt_A.ReadOutAutoRestoreProperties();
        _to_A._tSt_B.ReadOutAutoRestoreProperties();
        _to_A._tSt_A._tTt_A.ReadOutAutoRestoreProperties();
        _to_A._tSt_A._tTt_B.ReadOutAutoRestoreProperties();
        _to_A._tSt_B._tTt_A.ReadOutAutoRestoreProperties();
        _to_A._tSt_B._tTt_B.ReadOutAutoRestoreProperties();
        _done := TRUE;
        ProbeDoneWhen(_done);
        {endregion}
        {region "T318_AutoRestoreOnStateChange"}
    eTcoTaskTests.AutoRestoreOnStateChange:
        IF _plcCycleCounter = 1 THEN
            _to_A._tSt_A.ReadOutAutoRestoreProperties();
            _to_A._tSt_B.ReadOutAutoRestoreProperties();
            _to_A._tSt_A._tTt_A.ReadOutAutoRestoreProperties();
            _to_A._tSt_A._tTt_B.ReadOutAutoRestoreProperties();
            _to_A._tSt_B._tTt_A.ReadOutAutoRestoreProperties();
            _to_A._tSt_B._tTt_B.ReadOutAutoRestoreProperties();
            _to_A._tSt_A._tTt_A.ReadOutState();
            _to_A._tSt_B._tTt_B.ReadOutState();
        END_IF

        IF _plcCycleCounter = 2 THEN
            _to_A._tSt_A._tTt_A.Restore();
            _to_A._tSt_B._tTt_B.Restore();
            _to_A._tSt_A._tTt_A.ReadOutState();
            _to_A._tSt_B._tTt_B.ReadOutState();
        END_IF

        IF _plcCycleCounter = 3 THEN
            _to_A._tSt_A._tTt_A.Invoke();
            _to_A._tSt_B._tTt_B.Invoke();
            _to_A._tSt_A._tTt_A();
            _to_A._tSt_B._tTt_B();
            _to_A._tSt_A._tTt_A.ReadOutState();
            _to_A._tSt_B._tTt_B.ReadOutState();
        END_IF

        IF _plcCycleCounter = 4 THEN
            _to_A._tSt_A._tTt_A.Invoke();
            _to_A._tSt_A._tTt_A();
            _to_A._tSt_B._tTt_B();
            _to_A._tSt_A._tTt_A.ReadOutState();
            _to_A._tSt_B._tTt_B.ReadOutState();
        END_IF

        IF _plcCycleCounter = 5 THEN
            _to_A._tSt_A.ChangeState(_to_A._tSt_A._myState);
            _to_A._tSt_B.ChangeState(_to_A._tSt_B._myState);
            _to_A._tSt_A._tTt_A();
            _to_A._tSt_B._tTt_B();
            _to_A._tSt_A._tTt_A.ReadOutState();
            _to_A._tSt_B._tTt_B.ReadOutState();
        END_IF

        _done := _plcCycleCounter = 5;
        ProbeDoneWhen(_done);
        {endregion}
        {region "T320_InvokeDisabledTask"}
    eTcoTaskTests.InvokeDisabledTask:
        IF _plcCycleCounter = 1 THEN
            _to_A._sut_A.Restore();
            _to_A._sut_A.Disable();
            RETURN;
        END_IF

        IF NOT _done THEN
            _to_A._sut_A.Invoke();
            _to_A._sut_A();
            _to_A._sut_A.ReadOutState();
            _done := _plcCycleCounter >= 1 + _inUint;
            ProbeDoneWhen(_done);
        END_IF
        {endregion}
        {region "T321_DisableExecutingTask"}
    eTcoTaskTests.DisableExecutingTask:
        IF _plcCycleCounter = 1 THEN
            _to_A._sut_A.Enable();
            _to_A._sut_A.Invoke();
            _to_A._sut_A();
            _to_A._sut_A.ReadOutState();
            RETURN;
        END_IF

        IF _plcCycleCounter = 2 THEN
            _to_A._sut_A.Disable();
            _to_A._sut_A();
            _to_A._sut_A.ReadOutState();
            RETURN;
        END_IF

        IF _plcCycleCounter = 3 THEN
            _to_A._sut_A.Restore();
            _to_A._sut_A.Enable();
            _to_A._sut_A();
            _to_A._sut_A.ReadOutState();
            RETURN;
        END_IF

        IF _plcCycleCounter = 4 THEN
            _to_A._sut_A.Invoke();
            _to_A._sut_A();
            _to_A._sut_A.ReadOutState();
            RETURN;
        END_IF

        IF _plcCycleCounter = 5 THEN
            _to_A._sut_A.Restore();
            _to_A._sut_A();
            _to_A._sut_A.ReadOutState();
            _done := TRUE;
            ProbeDoneWhen(_done);
        END_IF
        {endregion}
        {region "T322_InvokeTaskThenDisable"}
    eTcoTaskTests.InvokeTaskThenDisable:
        _to_A._sut_A.Invoke();
        _to_A._sut_A.Disable();
        _to_A._sut_A();
        _to_A._sut_A.ReadOutState();
        _done := TRUE;
        ProbeDoneWhen(_done);
        {endregion}
        {region "T323_DisableTaskInErrorStateEnableAndTriggerAgain"}
    eTcoTaskTests.DisableTaskInErrorStateEnableAndTriggerAgain:
        IF _plcCycleCounter = 1 THEN
            _to_A._sut_A.Enable();
            _to_A._sut_A.Invoke();
            _to_A._sut_A();
            _to_A._sut_A.ReadOutState();
            RETURN;
        END_IF

        IF _plcCycleCounter = 2 THEN
            _to_A.CounterValue_A := _to_A.CounterValue_A + 5;
            _to_A._sut_A();
            _to_A._sut_A.ReadOutState();
            RETURN;
        END_IF

        IF _plcCycleCounter = 3 THEN
            _to_A._sut_A.Disable();
            _to_A._sut_A();
            _to_A._sut_A.ReadOutState();
            RETURN;
        END_IF

        IF _plcCycleCounter = 4 THEN
            _to_A._sut_A.Invoke();
            _to_A._sut_A();
            _to_A._sut_A.ReadOutState();
            RETURN;
        END_IF

        IF _plcCycleCounter = 5 THEN
            _to_A._sut_A.Restore();
            _to_A._sut_A.Invoke();
            _to_A._sut_A();
            _to_A._sut_A.ReadOutState();
            _done := TRUE;
            ProbeDoneWhen(_done);
        END_IF
        {endregion}
        {region "T330_ElapsedTypeMeasurement"}
    eTcoTaskTests.ElapsedTypeMeasurement:
        IF _plcCycleCounter = 1 THEN
            _to_A._sut_A.Restore();
            _to_A._sut_A.Enable();
            _to_A._sut_A.Invoke();
            RETURN;
        END_IF

        IF (_to_A._sut_A.Execute()) THEN
            _runElapsedTimer := TRUE;

            IF (_elapsedTimeTimer.Q) THEN
                _to_A._sut_A.DoneWhen(_elapsedTimeTimer.Q);
            END_IF;
        END_IF

        _done := _to_A._sut_A.Done;
        ProbeDoneWhen(_done);
        _elapsedTime := _to_A._sut_A.ElapsedTime;
        {endregion}
        {region "T340_TaskExecutingWithDoneAndErrorStatement"}
    eTcoTaskTests.TaskExecutingWithDoneAndErrorStatement:
        IF _plcCycleCounter = 1 THEN
            _to_A._sut_A.Restore();
            _to_A._sut_A.Enable();
            _to_A._sut_A.Invoke();
            _to_A._sut_A();
            _to_A._sut_A.ReadOutState();
            RETURN;
        END_IF

        _to_A._sut_A();
        _to_A._sut_A.DoneWhen(TRUE);
        _to_A._sut_A.ThrowWhen(TRUE);
        _to_A._sut_A.ReadOutState();
        _done := _to_A._sut_A.Done;
        ProbeDoneWhen(_done);
        {endregion}
        {region "T341_TaskExecutingWithErrorAndDoneStatement"}
    eTcoTaskTests.TaskExecutingWithErrorAndDoneStatement:
        IF _plcCycleCounter = 1 THEN
            _to_A._sut_A.Restore();
            _to_A._sut_A.Enable();
            _to_A._sut_A.Invoke();
            _to_A._sut_A();
            _to_A._sut_A.ReadOutState();
            RETURN;
        END_IF

        _to_A._sut_A();
        _to_A._sut_A.ThrowWhen(TRUE);
        _to_A._sut_A.DoneWhen(TRUE);
        _to_A._sut_A.ReadOutState();
        _done := _to_A._sut_A.Done;
        ProbeDoneWhen(_done);
        {endregion}
    eTcoTaskTests.TaskExecuteMethodNotCalled:
        _to_A._sut_A.Invoke().Done;
    eTcoTaskTests.TaskExecuteMethodCalled:
        _to_A._sut_A.Invoke().Done;
        _to_A._sut_A.Execute();
END_CASE
END_METHOD

METHOD INTERNAL ReadOutCycleCounters
_startCycles := THIS^.StartCycleCount;
_endCycles := THIS^.EndCycleCount;
_myIdentity := THIS^.Identity;
END_METHOD

END_FUNCTION_BLOCK

// ---- Tests/TcoTask/PlcExecuted/TcoTaskPlcTestObject.TcPOU
FUNCTION_BLOCK TcoTaskPlcTestObject EXTENDS TcoCore.TcoObject
VAR
    _myIdentity : ULINT;
    _myContextIdentity : ULINT;
    _myContextStartCount : ULINT;
    _myContextEndCount : ULINT;
    _myParentIdentity : ULINT;
    _sut_A : TcoTaskPlcTest(THIS^);
    _sut_B : TcoTaskPlcTest(THIS^);
    _tSt_A : TcoTaskPlcTestState(THIS^, eRestoreMode.AutoRestoreMembers);
    _tSt_B : TcoTaskPlcTestState(THIS^, eRestoreMode.None);
END_VAR

_sut_A();
_sut_B();

PROPERTY CounterValue_A : ULINT
GET
CounterValue_A := _sut_A.CounterValue;
END_GET
SET
_sut_A.CounterValue := CounterValue_A;
END_SET
END_PROPERTY

PROPERTY CounterValue_B : ULINT
GET
CounterValue_B := _sut_B.CounterValue;
END_GET
SET
_sut_B.CounterValue := CounterValue_B;
END_SET
END_PROPERTY

{attribute 'TcRpcEnable'}
METHOD INTERNAL ReadOutIdentities
_myIdentity := THIS^.Identity;
_myContextIdentity := THIS^.Context.Identity;
_myContextStartCount := THIS^.Context.StartCycleCount;
_myContextEndCount := THIS^.Context.EndCycleCount;
_myParentIdentity := THIS^.Parent.Identity;
END_METHOD

END_FUNCTION_BLOCK

// ---- Tests/TcoTask/PlcExecuted/TcoTaskPlcTest.TcPOU
FUNCTION_BLOCK TcoTaskPlcTest EXTENDS TcoCore.TcoTask
VAR
    _isBusy : BOOL;
    _isError : BOOL;
    _isDone : BOOL;
    _isReady : BOOL;
    _isInvokeRequestTrue : BOOL;
    _counterSetValue : ULINT;
    _counterValue : ULINT;
    _invokeCounter : ULINT;
    _executeCounter : ULINT;
    _doneCounter : ULINT;
    _invokeRisingEdgeCounter : ULINT;
    _executeRisingEdgeCounter : ULINT;
    _doneRisingEdgeCounter : ULINT;
    _previousState : eTaskState;
    _counterValuePV : ULINT;
    _myIdentity : ULINT;
    _myContextIdentity : ULINT;
    _myContextStartCount : ULINT;
    _myContextEndCount : ULINT;
    _myParentIdentity : ULINT;
    _autoRestoreByMyParentEnabled : BOOL;
    _onErrorCounter : ULINT;
    _whileErrorCounter : ULINT;
    _onStartCounter : ULINT;
END_VAR

IF (THIS^._taskState = eTaskState.Requested) THEN
    _invokeCounter := _invokeCounter + 1;
END_IF;

IF (THIS^._taskState = eTaskState.Requested AND _PreviousState <> eTaskState.Requested) THEN
    _counterValue := _counterSetValue;
    _counterValuePV := _counterValue;
    _invokeRisingEdgeCounter := _invokeRisingEdgeCounter + 1;
END_IF

IF (THIS^._taskState = eTaskState.Busy AND _previousState <> eTaskState.Busy) THEN
    _executeRisingEdgeCounter := _executeRisingEdgeCounter + 1;
END_IF

_previousState := THIS^._taskState;

IF (Execute()) THEN
    _executeCounter := _executeCounter + 1;
    _counterValue := _counterValue - 1;
    DoneWhen(_counterValue <= 0);
    ThrowWhen(ABS(_counterValuePV - _counterValue) > 1);
    _CounterValuePV := _counterValue;
END_IF

IF (THIS^._taskState = eTaskState.Done) THEN
    _doneCounter := _doneCounter + 1;
END_IF;

IF (THIS^._taskState = eTaskState.Done AND _previousState <> eTaskState.Done) THEN
    _doneRisingEdgeCounter := _doneRisingEdgeCounter + 1;
END_IF

PROPERTY CounterValue : ULINT
GET
CounterValue := _counterValue;
END_GET
SET
_counterValue := CounterValue;
END_SET
END_PROPERTY

METHOD INTERNAL Disable
THIS^.Enabled := FALSE;
END_METHOD

METHOD INTERNAL Enable
THIS^.Enabled := TRUE;
END_METHOD

METHOD INTERNAL GetMessage : STRING
GetMessage := SUPER^._messenger._mime.Text;
END_METHOD

METHOD PROTECTED OnError
_onErrorCounter := _onErrorCounter + 1;
END_METHOD

METHOD PROTECTED OnStart
_onStartCounter := _onStartCounter + 1;
END_METHOD

METHOD INTERNAL PostMessage
VAR_INPUT
    Message : STRING;
END_VAR
THIS^.Messenger.Post(Message, eMessageCategory.Error);
END_METHOD

{attribute 'TcRpcEnable'}
METHOD INTERNAL ReadOutAutoRestoreProperties
_autoRestoreByMyParentEnabled := THIS^.AutoRestorable;
END_METHOD

{attribute 'TcRpcEnable'}
METHOD INTERNAL ReadOutIdentities
_myIdentity := THIS^.Identity;
_myContextIdentity := THIS^.Context.Identity;
_myContextStartCount := THIS^.Context.StartCycleCount;
_myContextEndCount := THIS^.Context.EndCycleCount;
_myParentIdentity := THIS^.Parent.Identity;
END_METHOD

{attribute 'TcRpcEnable'}
METHOD INTERNAL ReadOutState
_isBusy := THIS^.Busy;
_isError := THIS^.Error;
_isDone := THIS^.Done;
_isReady := THIS^.Ready;
_isInvokeRequestTrue := THIS^._invokeRequest;
END_METHOD

{attribute 'TcRpcEnable'}
METHOD INTERNAL SetInvokeRequest
THIS^._invokeRequest := TRUE;
END_METHOD

{attribute 'TcRpcEnable'}
METHOD INTERNAL SetPreviousStateToReady
THIS^._previousState := eTaskState.Ready;
END_METHOD

(*~
    <docu>
        <summary>
            Executes until task is in ```Error``` state .
        </summary>
    </docu>
~*)
METHOD PROTECTED WhileError
_whileErrorCounter := _whileErrorCounter + 1;
END_METHOD

END_FUNCTION_BLOCK

// ---- Tests/TcoTask/PlcExecuted/TcoTaskPlcTestState.TcPOU
FUNCTION_BLOCK TcoTaskPlcTestState EXTENDS TcoState
VAR
    _myIdentity : ULINT;
    _myContextIdentity : ULINT;
    _myContextStartCount : ULINT;
    _myContextEndCount : ULINT;
    _myParentIdentity : ULINT;
    _myState : INT;
    _tTt_A : TcoTaskPlcTest(THIS^);
    _tTt_B : TcoTaskPlcTest(THIS^);
    _onStateChangeCounter : INT;
    _autoRestoreToMyChildsEnabled : BOOL;
    _autoRestoreByMyParentEnabled : BOOL;
END_VAR

METHOD PROTECTED OnStateChange
VAR_INPUT
    PreviousState : INT;
    NewState : INT;
END_VAR
VAR
    message : STRING;
END_VAR
_onStateChangeCounter := _onStateChangeCounter + 1;
message := CONCAT('My state has been change from ', INT_TO_STRING(PreviousState));
message := CONCAT(message, ' to the new state ');
message := CONCAT(message, INT_TO_STRING(NewState));
message := CONCAT(message, '.');
THIS^.Messenger.Post(message, eMessageCategory.Debug);
SUPER^.OnStateChange(PreviousState, NewState);
END_METHOD

{attribute 'TcRpcEnable'}
METHOD INTERNAL ReadOutAutoRestoreProperties
_autoRestoreToMyChildsEnabled := THIS^.IsAutoRestoreEnabled;
_autoRestoreByMyParentEnabled := THIS^.AutoRestorable;
END_METHOD

{attribute 'TcRpcEnable'}
METHOD INTERNAL ReadOutIdentities
_myIdentity := THIS^.Identity;
_myContextIdentity := THIS^.Context.Identity;
_myParentIdentity := THIS^.Parent.Identity;
_myContextStartCount := THIS^.Context.StartCycleCount;
_myContextEndCount := THIS^.Context.EndCycleCount;
END_METHOD

{attribute 'TcRpcEnable'}
METHOD INTERNAL ReadOutState
_myState := THIS^.State;
THIS^._tTt_A.ReadOutState();
THIS^._tTt_B.ReadOutState();
END_METHOD

{attribute 'TcRpcEnable'}
METHOD INTERNAL TriggerChangeState
VAR_INPUT
    NewState : INT;
END_VAR
THIS^.ChangeState(NewState);
END_METHOD

{attribute 'TcRpcEnable'}
METHOD INTERNAL TriggerChangeStateWithObjectRestore
VAR_INPUT
    NewState : INT;
END_VAR
THIS^.ChangeState(NewState).RestoreObject(THIS^._tTt_A).RestoreObject(THIS^._tTt_B);
END_METHOD

{attribute 'TcRpcEnable'}
METHOD INTERNAL TriggerRestore
THIS^.Restore();
END_METHOD

{attribute 'TcRpcEnable'}
METHOD INTERNAL TriggerTaskInvoke
THIS^._tTt_A.Invoke();
THIS^._tTt_B.Invoke();
END_METHOD

END_FUNCTION_BLOCK

// ---- Tests/TcoToggleTask/TcoToggleTaskTestContext.TcPOU
FUNCTION_BLOCK TcoToggleTaskTestContext EXTENDS TcoCore._internals_TcoContext
VAR
    _sut : TcoToggleTaskTests(THIS^, TRUE);
    _bool : BOOL;
    _string : STRING;
    _done : BOOL;
END_VAR

METHOD PROTECTED Main
CASE _testId OF
    eTcoToggleTaskTests.Reinit:
        _sut.FB_init(TRUE,
            FALSE,
            THIS^,
            _bool);

        _done := TRUE;
    eTcoToggleTaskTests.CleanUp:
        IF NOT _done THEN
            _sut._messenger.Clear();
            _done := TRUE;
        END_IF
    eTcoToggleTaskTests.Message:
        IF NOT _done THEN
            _sut.Messenger.Error(_string);
            _done := TRUE;
        END_IF
    eTcoToggleTaskTests.TriggerToggleWhileRunNotCalled:
        IF NOT _done THEN
            _sut._messenger.Clear();
            _sut.Toggle();
            _done := TRUE;
        END_IF
    eTcoToggleTaskTests.TriggerToggleWhileDisabled:
        IF NOT _done THEN
            _sut.Run();
            _sut._messenger.Clear();
            _sut.Enabled := FALSE;
            _sut.Toggle();
            _done := TRUE;
        END_IF
    eTcoToggleTaskTests.TriggerToggleWhileEnabled:
        IF NOT _done THEN
            _sut.Run();
            _sut._messenger.Clear();
            _sut.Enabled := TRUE;
            _sut.Toggle();
            _done := TRUE;
        END_IF
    eTcoToggleTaskTests.TriggerOnWhileRunNotCalled:
        IF NOT _done THEN
            _sut._messenger.Clear();
            _sut.On();
            _done := TRUE;
        END_IF
    eTcoToggleTaskTests.TriggerOnWhileDisabled:
        IF NOT _done THEN
            _sut.Run();
            _sut._messenger.Clear();
            _sut.Enabled := FALSE;
            _sut.On();
            _done := TRUE;
        END_IF
    eTcoToggleTaskTests.TriggerOnWhileEnabled:
        IF NOT _done THEN
            _sut.Run();
            _sut._messenger.Clear();
            _sut.Enabled := TRUE;
            _sut.On();
            _done := TRUE;
        END_IF
    eTcoToggleTaskTests.TriggerOffWhileRunNotCalled:
        IF NOT _done THEN
            _sut._messenger.Clear();
            _sut.Toggle();
            _done := TRUE;
        END_IF
    eTcoToggleTaskTests.TriggerOffWhileDisabled:
        IF NOT _done THEN
            _sut.Run();
            _sut._messenger.Clear();
            _sut.Enabled := FALSE;
            _sut.Off();
            _done := TRUE;
        END_IF
    eTcoToggleTaskTests.TriggerOffWhileEnabled:
        IF NOT _done THEN
            _sut.Run();
            _sut._messenger.Clear();
            _sut.Enabled := TRUE;
            _sut.Off();
            _done := TRUE;
        END_IF
END_CASE
END_METHOD

END_FUNCTION_BLOCK

// ---- Tests/TcoToggleTask/TcoToggleTaskTests.TcPOU
FUNCTION_BLOCK TcoToggleTaskTests EXTENDS TcoCore.TcoToggleTask
VAR
    _isOn : BOOL;
    _isOff : BOOL;
    _isEnabled : BOOL;
    _isToggleRequestTrue : BOOL;
    _counterValue : ULINT;
    _counterValuePV : ULINT;
    _toggleCounter : ULINT;
    _runCounter : ULINT;
    _onFtrigCounter : ULINT;
    _onRtrigCounter : ULINT;
    _onCounter : ULINT;
    _offCounter : ULINT;
    _onStateChangeCounter : ULINT;
    _taskOnCounter : ULINT;
    _taskOffCounter : ULINT;
    _stateChangedCounter : ULINT;
    _previousState : BOOL;
    _myIdentity : ULINT;
    _myContextIdentity : ULINT;
    _myContextStartCount : ULINT;
    _myContextEndCount : ULINT;
    _myParentIdentity : ULINT;
END_VAR

ExecutionBody();

METHOD INTERNAL Disable
THIS^.Enabled := FALSE;
END_METHOD

METHOD INTERNAL Enable
THIS^.Enabled := TRUE;
END_METHOD

{attribute 'TcRpcEnable'}
METHOD INTERNAL ExecutionBody
Run();
_runCounter := _runCounter + 1;

IF _previousState <> THIS^.State THEN
    _stateChangedCounter := _stateChangedCounter + 1;
END_IF;

_previousState := THIS^.State;
END_METHOD

{attribute 'TcRpcEnable'}
METHOD INTERNAL GetMessage : STRING
GetMessage := SUPER^._messenger._mime.Text;
END_METHOD

METHOD PROTECTED Main
VAR
END_VAR
END_METHOD

(*~
    <docu>
        <summary>
            Executes when toggle task changes its state from '''TRUE''' to '''FALSE'''.
        </summary>
    </docu>
~*)
METHOD PROTECTED OnFtrig
_onFtrigCounter := _onFtrigCounter + 1;
END_METHOD

(*~
    <docu>
        <summary>
            Executes when toggle task changes its state from '''FALSE''' to '''TRUE'''.
        </summary>
    </docu>
~*)
METHOD PROTECTED OnRtrig
_onRtrigCounter := _onRtrigCounter + 1;
END_METHOD

(*~
    <docu>
        <summary>
            Executes when toggle task changes its state .
        </summary>
    </docu>
~*)
METHOD PROTECTED OnStateChange
_onStateChangeCounter := _onStateChangeCounter + 1;
END_METHOD

{attribute 'TcRpcEnable'}
METHOD INTERNAL PostMessage
VAR_INPUT
    Message : STRING;
END_VAR
THIS^.Messenger.Post(Message, eMessageCategory.Error);
END_METHOD

{attribute 'TcRpcEnable'}
METHOD INTERNAL ReadOutIdentities
_myIdentity := THIS^.Identity;
_myContextIdentity := THIS^.Context.Identity;
_myContextStartCount := THIS^.Context.StartCycleCount;
_myContextEndCount := THIS^.Context.EndCycleCount;
_myParentIdentity := THIS^.Parent.Identity;
END_METHOD

{attribute 'TcRpcEnable'}
METHOD INTERNAL ReadOutState
_isOn := THIS^.IsOn;
_isOff := THIS^.IsOff;
_isEnabled := THIS^.Enabled;
_isToggleRequestTrue := THIS^._toggleRequest;
END_METHOD

{attribute 'TcRpcEnable'}
METHOD INTERNAL SetPreviousState
VAR_INPUT
    inValue : BOOL;
END_VAR
THIS^._previousState := inValue;
END_METHOD

{attribute 'TcRpcEnable'}
METHOD INTERNAL SetState
VAR_INPUT
    inState : BOOL;
END_VAR
THIS^._state := inState;
END_METHOD

{attribute 'TcRpcEnable'}
METHOD INTERNAL SetToggleRequest
THIS^._toggleRequest := TRUE;
END_METHOD

(*~
    <docu>
        <summary>
            Executes when toggle task is in ```Off``` state .
        </summary>
    </docu>
~*)
METHOD PROTECTED TaskOff
_taskOffCounter := _taskOffCounter + 1;
_counterValue := _counterValue - 1;
_CounterValuePV := _counterValue;
END_METHOD

(*~
    <docu>
        <summary>
            Executes when toggle task is in  ```On``` state .
        </summary>
    </docu>
~*)
METHOD PROTECTED TaskOn
_taskOnCounter := _taskOnCounter + 1;
_counterValue := _counterValue + 1;
_CounterValuePV := _counterValue;
END_METHOD

{attribute 'TcRpcEnable'}
METHOD INTERNAL TriggerOff
THIS^.Off();
_offCounter := _offCounter + 1;
END_METHOD

{attribute 'TcRpcEnable'}
METHOD INTERNAL TriggerOn
THIS^.On();
_onCounter := _onCounter + 1;
END_METHOD

{attribute 'TcRpcEnable'}
METHOD INTERNAL TriggerToggle
THIS^.Toggle();
_toggleCounter := _toggleCounter + 1;
END_METHOD

END_FUNCTION_BLOCK

// ---- Tests/TcoComponent/PlcExecuted/TcoComponentTestContext.TcPOU
FUNCTION_BLOCK TcoComponentTestContext EXTENDS TcoCore._internals_TcoContext
VAR
    _sut : TestComponent(THIS^);
    {attribute addProperty Name "--Some IO signal"}
    _signal : BOOL;
END_VAR

METHOD PROTECTED Main
CASE _testId OF
    eTcoComponentTests.GetSignalInfo:
        _sut(_signal := _signal);
END_CASE
END_METHOD

END_FUNCTION_BLOCK

// ---- Tests/TcoComponent/PlcExecuted/TestComponent.TcPOU
FUNCTION_BLOCK TestComponent EXTENDS TcoCore.TcoComponent
VAR_IN_OUT
    _signal : BOOL;
END_VAR
VAR
    _signalInfo : TcoCore.TcoSignalInfo;
END_VAR

_signalInfo.GetSignalInfo(SIZEOF(_signal), ADR(_signal));

(*~
    <docu>
        <summary>
            Restores this instance to the Ready state. Can be called explicitly or from within one of the restore mechanisms.
        </summary>
    </docu>
~*)
METHOD Restore : ITcoRestorable
END_METHOD

(*~
    <docu>
        <summary>
            Custom service (manual, maintenance) logic.
            This method must be implemented in derived class.
        </summary>
    </docu>
~*)
METHOD PROTECTED ServiceMode
END_METHOD

END_FUNCTION_BLOCK

// ---- Tests/TcoRemoteTask/PlcExecuted/TcoRemoteTaskTestContext.TcPOU
FUNCTION_BLOCK TcoRemoteTaskTestContext EXTENDS TcoCore._internals_TcoContext
VAR
    _sut : TcoRemoteTaskTest(THIS^);
    _invokeInitializedCSharpMethodDone : BOOL;
    _invokeNotInitializedCSharpMethodDone : BOOL;
    _exceptionInMethodWillResultInExceptionDone : BOOL;
    _sharedVariable : INT;
END_VAR

METHOD PROTECTED Main
CASE _testId OF
    0:
        _invokeInitializedCSharpMethodDone := FALSE;
        _invokeNotInitializedCSharpMethodDone := FALSE;
        _exceptionInMethodWillResultInExceptionDone := FALSE;
    eTcoRemoteTaskTests.RestoreTasks:
        _sut._invokeInitializedCSharpMethod.Restore();
        _sut._invokeNotInitializedCSharpMethod.Restore();
        _sut._exceptionInMethodWillResultInException.Restore();
    eTcoRemoteTaskTests.InvokeInitializedCSharpMethod:
        _invokeInitializedCSharpMethodDone := _sut._invokeInitializedCSharpMethod.Invoke().Done;
    eTcoRemoteTaskTests.InvokeNotInitializedCSharpMethod:
        _invokeNotInitializedCSharpMethodDone := _sut._invokeNotInitializedCSharpMethod.Invoke().Error;
    eTcoRemoteTaskTests.ExceptionInMethodWillResultInException:
        _exceptionInMethodWillResultInExceptionDone := _sut._exceptionInMethodWillResultInException.Invoke().Error;
END_CASE

_sut();
END_METHOD

END_FUNCTION_BLOCK

// ---- Tests/TcoRemoteTask/PlcExecuted/TcoRemoteTaskTest.TcPOU
FUNCTION_BLOCK TcoRemoteTaskTest EXTENDS TcoCore.TcoObject
VAR
    _invokeInitializedCSharpMethod : TcoCore.TcoRemoteTask(THIS^);
    _invokeNotInitializedCSharpMethod : TcoCore.TcoRemoteTask(THIS^);
    _exceptionInMethodWillResultInException : TcoCore.TcoRemoteTask(THIS^);
END_VAR

_invokeInitializedCSharpMethod();
_invokeNotInitializedCSharpMethod();
_exceptionInMethodWillResultInException();

END_FUNCTION_BLOCK

// ---- Tests/TcoSequencer/PlcExecuted/TcoSequencerTestContext.TcPOU
FUNCTION_BLOCK TcoSequencerTestContext EXTENDS TcoCore._internals_TcoContext
VAR
    _sut_A : TcoSequencerTestType(THIS^, eRestoreMode.AutoRestoreMembers);
    _sut_N : TcoSequencerTestType(THIS^, eRestoreMode.None);
    _elapsedTimeETA : TIME;
    _elapsedTime : TIME;
    _runElapsedTimer : BOOL;
    _elapsedTimeTimer : Tc2_Standard.TON;
    _runOneStep : BOOL;
    _runAllSteps : BOOL;
    _finishStep : BOOL;
    _stepId : INT;
    _enabled : BOOL;
    _stepDescription : STRING(254);
    _currentStepId : INT;
    _currentStepDescription : STRING(254);
    _totalStepNumber : UINT;
    _reqStep : INT;
    _reqStepNotExists : INT;
    _done : BOOL;
    _arranged : BOOL;
    _startCycles : ULINT;
    _endCycles : ULINT;
    _myIdentity : ULINT;
    _initReqStepCycle : UINT;
    _cycles : UINT;
    _cyclicCycles : UINT;
    _stepInEvents : UINT;
END_VAR

{attribute 'TcRpcEnable'}
METHOD _ClearPlcCycleCounter
ClearPlcCycleCounter();
END_METHOD

METHOD PROTECTED Main
VAR
    i : INT;
END_VAR
_elapsedTimeTimer(IN := _runElapsedTimer, PT := _elapsedTimeETA);

CASE _testId OF
    {region "CallSequencerBodiesOnly"}
    eTcoSequencerTests.CallSequencerBodiesOnly:
        _sut_A.TcoSequencerTest := eTcoSequencerTests.CallSequencerBodiesOnly;
        _sut_N.TcoSequencerTest := eTcoSequencerTests.CallSequencerBodiesOnly;
        _sut_A.Run();
        _sut_N.Run();
        {endregion}
        {region "RestoreSequencers"}
    eTcoSequencerTests.RestoreSequencers:
        IF NOT _arranged THEN
            _sut_A.Restore();
            _sut_N.Restore();
            _arranged := _sut_A._restoringSequence AND _sut_N._restoringSequence;
        END_IF

        IF _arranged AND NOT _done THEN
            _sut_A.TcoSequencerTest := eTcoSequencerTests.RestoreSequencers;
            _sut_N.TcoSequencerTest := eTcoSequencerTests.RestoreSequencers;
            _sut_A.Run();
            _sut_N.Run();

            _done :=
                NOT _sut_A._restoringSequence AND NOT _sut_N._restoringSequence AND NOT _sut_A._sequencerHasError AND NOT _sut_N._sequencerHasError;
        END_IF

        ProbeDoneWhen(_done);
        {endregion}
        {region "T500_NumberOfStepsCount"}
    eTcoSequencerTests.NumberOfStepsCount:
        IF NOT _arranged THEN
            _sut_A.SetCyclicMode(); //Set sequencer into the cyclic mode
            _sut_N.SetCyclicMode(); //Set sequencer into the cyclic mode
            _sut_A.SetSequenceAsChecked(); //Set sequence as checked, so no StepID uniqueness is performed on next sequence execution
            _sut_N.SetSequenceAsChecked(); //Set sequence as checked, so no StepID uniqueness is performed on next sequence execution
            _sut_A.ClearNumberOfSteps(); //Clear internal flow step counters, so number of steps is going to be counted again on next sequence run
            _sut_N.ClearNumberOfSteps(); //Clear internal flow step counters, so number of steps is going to be counted again on next sequence run

            _sut_A.SetCurrentStep(_currentStepId,
                _currentStepDescription); //Set the StepId so as the StepDescription to the current step of the sequencer

            _sut_N.SetCurrentStep(_currentStepId,
                _currentStepDescription); //Set the StepId so as the StepDescription to the current step of the sequencer

            _sut_A.SaveNumberOfStepsInSequence();
            _sut_N.SaveNumberOfStepsInSequence();
            _sut_A.TcoSequencerTest := eTcoSequencerTests.NumberOfStepsCount;
            _sut_N.TcoSequencerTest := eTcoSequencerTests.NumberOfStepsCount;
            _sut_A.TotalStepNumber := _totalStepNumber;
            _sut_N.TotalStepNumber := _totalStepNumber;
            _sut_A.FinishStep := FALSE;
            _sut_N.FinishStep := FALSE;
            _arranged := TRUE;
            RETURN;
        END_IF

        IF NOT _done THEN
            _sut_A.Run();
            _sut_N.Run();
            _sut_A.SaveNumberOfStepsInSequence();
            _sut_N.SaveNumberOfStepsInSequence();
            _done := TRUE;
        END_IF

        IF _done THEN
            ProbeDoneWhen(_done);
        END_IF
        {endregion}
        {region "T501_ExecutionInOnePLCcycle"}
    eTcoSequencerTests.ExecutionInOnePLCcycle:
        _sut_A.TcoSequencerTest := eTcoSequencerTests.ExecutionInOnePLCcycle;
        _sut_N.TcoSequencerTest := eTcoSequencerTests.ExecutionInOnePLCcycle;
        _sut_A.SetCyclicMode(); //Set sequencer into the cyclic mode
        _sut_N.SetCyclicMode(); //Set sequencer into the cyclic mode
        _sut_A.TotalStepNumber := _totalStepNumber;
        _sut_N.TotalStepNumber := _totalStepNumber;
        _sut_A.Run();
        _sut_N.Run();
        _done := TRUE;
        ProbeDoneWhen(_done);
        {endregion}
        {region "T502_OnStepCompleted"}
    eTcoSequencerTests.OnStepCompleted:
        _sut_A.TcoSequencerTest := eTcoSequencerTests.OnStepCompleted;
        _sut_N.TcoSequencerTest := eTcoSequencerTests.OnStepCompleted;
        _sut_A.TotalStepNumber := _totalStepNumber;
        _sut_N.TotalStepNumber := _totalStepNumber;
        _sut_A.Run();
        _sut_N.Run();
        _sut_A.SaveNumberOfStepsInSequence();
        _sut_N.SaveNumberOfStepsInSequence();
        _done := TRUE;
        ProbeDoneWhen(_done);
        {endregion}
        {region "T503_OnSequenceCompleted"}
    eTcoSequencerTests.OnSequenceCompleted:
        _sut_A.TcoSequencerTest := eTcoSequencerTests.OnSequenceCompleted;
        _sut_N.TcoSequencerTest := eTcoSequencerTests.OnSequenceCompleted;
        _sut_A.TotalStepNumber := _totalStepNumber;
        _sut_N.TotalStepNumber := _totalStepNumber;
        _sut_A.Run();
        _sut_N.Run();
        _done := TRUE;
        ProbeDoneWhen(_done);
        {endregion}
        {region "T504_RestoreChildBetweenSteps"}
    eTcoSequencerTests.RestoreChildBetweenSteps:
        IF NOT _arranged THEN
            _sut_A.TcoSequencerTest := eTcoSequencerTests.RestoreChildBetweenSteps;
            _sut_N.TcoSequencerTest := eTcoSequencerTests.RestoreChildBetweenSteps;
            _sut_A.TotalStepNumber := _totalStepNumber;
            _sut_N.TotalStepNumber := _totalStepNumber;
            _arranged := TRUE;
            RETURN;
        END_IF;

        _sut_A.Run();
        _sut_N.Run();
        _done := TRUE;
        ProbeDoneWhen(_done);
        {endregion}
        {region "T505_OnStateChangeWithRestoreCallInside"}
    eTcoSequencerTests.OnStateChangeWithRestoreCallInside:
        IF NOT _arranged THEN
            _sut_A.SetCyclicMode(); //Set sequencer into the cyclic mode
            _sut_N.SetCyclicMode(); //Set sequencer into the cyclic mode
            _sut_A.SetSequenceAsChecked(); //Set sequence as checked, so no StepID uniqueness is performed on next sequence execution
            _sut_N.SetSequenceAsChecked(); //Set sequence as checked, so no StepID uniqueness is performed on next sequence execution
            _sut_A.SetNumberOfSteps(_totalStepNumber); //Set numberOfSteps to the testing instance
            _sut_N.SetNumberOfSteps(_totalStepNumber); //Set numberOfSteps to the testing instance
            _sut_A.TcoSequencerTest := eTcoSequencerTests.OnStateChangeWithRestoreCallInside;
            _sut_N.TcoSequencerTest := eTcoSequencerTests.OnStateChangeWithRestoreCallInside;
            _sut_A.TotalStepNumber := _totalStepNumber;
            _sut_N.TotalStepNumber := _totalStepNumber;
            _sut_A.FinishStep := FALSE;
            _sut_N.FinishStep := FALSE;
            _plcCycleCounter := 0;
            _arranged := TRUE;
            RETURN;
        END_IF

        IF NOT _done THEN
            IF _plcCycleCounter = 1 THEN
                _sut_A.CallRestoreInOnStateChange := FALSE;
                _sut_N.CallRestoreInOnStateChange := FALSE;
            ELSE
                _sut_A.CallRestoreInOnStateChange := TRUE;
                _sut_N.CallRestoreInOnStateChange := TRUE;
                _sut_A.FinishStep := TRUE;
                _sut_N.FinishStep := TRUE;
            END_IF

            _sut_A.Run();
            _sut_N.Run();
        END_IF

        _done := _plcCycleCounter >= 2;

        IF _done THEN
            _sut_A.CallRestoreInOnStateChange := FALSE;
            _sut_N.CallRestoreInOnStateChange := FALSE;
            ProbeDoneWhen(_done);
        END_IF
        {endregion}
        {region "T506_MinStepId"}
    eTcoSequencerTests.MinStepId:
        IF NOT _arranged THEN
            _sut_A.SetCyclicMode(); //Set sequencer into the cyclic mode
            _sut_N.SetCyclicMode(); //Set sequencer into the cyclic mode
            _sut_A.SetSequenceAsChecked(); //Set sequence as checked, so no StepID uniqueness is performed on next sequence execution
            _sut_N.SetSequenceAsChecked(); //Set sequence as checked, so no StepID uniqueness is performed on next sequence execution
            _sut_A.SetNumberOfSteps(_totalStepNumber); //Set numberOfSteps to the testing instance
            _sut_N.SetNumberOfSteps(_totalStepNumber); //Set numberOfSteps to the testing instance
            _sut_A.TcoSequencerTest := eTcoSequencerTests.MinStepId;
            _sut_N.TcoSequencerTest := eTcoSequencerTests.MinStepId;
            _sut_A.TotalStepNumber := _totalStepNumber;
            _sut_N.TotalStepNumber := _totalStepNumber;
            _sut_A.FinishStep := FALSE;
            _sut_N.FinishStep := FALSE;
            _plcCycleCounter := 0;
            _arranged := TRUE;
            RETURN;
        END_IF

        IF NOT _done THEN
            _sut_A.StepId := _currentStepId;
            _sut_N.StepId := _currentStepId;
            _sut_A.Run();
            _sut_N.Run();
        END_IF

        _done := TRUE;
        ProbeDoneWhen(_done);
        {endregion}
        {region "T507_MaxStepId"}
    eTcoSequencerTests.MaxStepId:
        IF NOT _arranged THEN
            _sut_A.SetCyclicMode(); //Set sequencer into the cyclic mode
            _sut_N.SetCyclicMode(); //Set sequencer into the cyclic mode
            _sut_A.SetSequenceAsChecked(); //Set sequence as checked, so no StepID uniqueness is performed on next sequence execution
            _sut_N.SetSequenceAsChecked(); //Set sequence as checked, so no StepID uniqueness is performed on next sequence execution
            _sut_A.SetNumberOfSteps(_totalStepNumber); //Set numberOfSteps to the testing instance
            _sut_N.SetNumberOfSteps(_totalStepNumber); //Set numberOfSteps to the testing instance
            _sut_A.TcoSequencerTest := eTcoSequencerTests.MaxStepId;
            _sut_N.TcoSequencerTest := eTcoSequencerTests.MaxStepId;
            _sut_A.TotalStepNumber := _totalStepNumber;
            _sut_N.TotalStepNumber := _totalStepNumber;
            _sut_A.FinishStep := FALSE;
            _sut_N.FinishStep := FALSE;
            _plcCycleCounter := 0;
            _arranged := TRUE;
            RETURN;
        END_IF

        IF NOT _done THEN
            _sut_A.StepId := _currentStepId;
            _sut_N.StepId := _currentStepId;
            _sut_A.Run();
            _sut_N.Run();
        END_IF

        _done := TRUE;
        ProbeDoneWhen(_done);
        {endregion}
        {region "T508_RequestStepToFirstStepWithStepId0"}
    eTcoSequencerTests.RequestStepToFirstStepWithStepId0:
        IF NOT _arranged THEN
            _sut_A.SetCyclicMode(); //Set sequencer into the cyclic mode
            _sut_N.SetCyclicMode(); //Set sequencer into the cyclic mode
            _sut_A.SetSequenceAsChecked(); //Set sequence as checked, so no StepID uniqueness is performed on next sequence execution
            _sut_N.SetSequenceAsChecked(); //Set sequence as checked, so no StepID uniqueness is performed on next sequence execution
            _sut_A.SetNumberOfSteps(_totalStepNumber); //Set numberOfSteps to the testing instance
            _sut_N.SetNumberOfSteps(_totalStepNumber); //Set numberOfSteps to the testing instance
            _sut_A.TcoSequencerTest := eTcoSequencerTests.RequestStepToFirstStepWithStepId0;
            _sut_N.TcoSequencerTest := eTcoSequencerTests.RequestStepToFirstStepWithStepId0;
            _sut_A.TotalStepNumber := _totalStepNumber;
            _sut_N.TotalStepNumber := _totalStepNumber;
            _sut_A.FinishStep := TRUE;
            _sut_N.FinishStep := TRUE;
            _plcCycleCounter := 0;
            _arranged := TRUE;
            RETURN;
        END_IF

        IF NOT _done THEN
            IF _plcCycleCounter > 1 THEN
                _sut_A.FinishStep := FALSE;
                _sut_N.FinishStep := FalsE;
            END_IF

            _sut_A.Run();
            _sut_N.Run();
        END_IF

        _done := _plcCycleCounter > 1;
        ProbeDoneWhen(_done);
        {endregion}
        {region "T509_RequestStep"}
    eTcoSequencerTests.RequestStep:
        IF NOT _arranged THEN
            _sut_A.SetCyclicMode(); //Set sequencer into the cyclic mode
            _sut_N.SetCyclicMode(); //Set sequencer into the cyclic mode
            _sut_A.SetSequenceAsChecked(); //Set sequence as checked, so no StepID uniqueness is performed on next sequence execution
            _sut_N.SetSequenceAsChecked(); //Set sequence as checked, so no StepID uniqueness is performed on next sequence execution
            _sut_A.SetNumberOfSteps(10); //Set numberOfSteps to the testing instance
            _sut_N.SetNumberOfSteps(10); //Set numberOfSteps to the testing instance
            _sut_A.TcoSequencerTest := eTcoSequencerTests.RequestStep;
            _sut_N.TcoSequencerTest := eTcoSequencerTests.RequestStep;
            _plcCycleCounter := 0;
            _arranged := TRUE;
            RETURN;
        END_IF

        IF NOT _done THEN
            _sut_A.SequenceRun := _plcCycleCounter;
            _sut_N.SequenceRun := _plcCycleCounter;
            _sut_A.Run();
            _sut_N.Run();
        END_IF

        _done := _plcCycleCounter >= 3;
        ProbeDoneWhen(_done);
        {endregion}
        {region "T510_CheckStepIdUniqueness"}
    eTcoSequencerTests.CheckStepIdUniqueness:
        IF NOT _arranged THEN
            _sut_A.SetCyclicMode(); //Set sequencer into the cyclic mode
            _sut_N.SetCyclicMode(); //Set sequencer into the cyclic mode
            _sut_A.SetSequenceAsNotChecked(); //Set sequence as not checked, so StepId uniqueness is going to be performed on next sequence run
            _sut_N.SetSequenceAsNotChecked(); //Set sequence as not checked, so StepId uniqueness is going to be performed on next sequence run
            _sut_A.ClearNumberOfSteps(); //Clear internal step counters, so number of steps is going to be counted again on next sequence run
            _sut_N.ClearNumberOfSteps(); //Clear internal step counters, so number of steps is going to be counted again on next sequence run
            _sut_A.Enabled := TRUE;
            _sut_A.RunOneStep := FALSE;
            _sut_A.RunAllSteps := TRUE;
            _sut_A.FinishStep := TRUE;
            _sut_N.Enabled := TRUE;
            _sut_N.RunOneStep := FALSE;
            _sut_N.RunAllSteps := TRUE;
            _sut_N.FinishStep := TRUE;
            _sut_A.SetCurrentStep(inStepID := _currentStepId, inStepDescription := _currentStepDescription);
            _sut_N.SetCurrentStep(inStepID := _currentStepId, inStepDescription := _currentStepDescription);
            _sut_A.TcoSequencerTest := eTcoSequencerTests.CheckStepIdUniqueness;
            _sut_N.TcoSequencerTest := eTcoSequencerTests.CheckStepIdUniqueness;
            _sut_A.SaveNumberOfStepsInSequence();
            _sut_N.SaveNumberOfStepsInSequence();
            _plcCycleCounter := 0;
            _arranged := TRUE;
            RETURN;
        END_IF

        IF NOT _done THEN
            _sut_A.Run();
            _sut_N.Run();
            _sut_A.SaveNumberOfStepsInSequence();
            _sut_N.SaveNumberOfStepsInSequence();
        END_IF

        _done := _plcCycleCounter >= 2;
        ProbeDoneWhen(_done);
        {endregion}
        {region "T512_RestoreAlreadyCheckedSequence"}
    eTcoSequencerTests.RestoreAlreadyCheckedSequence:
        _sut_A.Restore();
        _sut_N.Restore();
        _sut_A.SaveNumberOfStepsInSequence();
        _sut_N.SaveNumberOfStepsInSequence();
        _done := TRUE;
        ProbeDoneWhen(_done);
        {endregion}
        {region "T513_CheckStepIdUniqueness"}
    eTcoSequencerTests.NotUniqueStepId:
        IF NOT _arranged THEN
            _sut_A.Enabled := TRUE;
            _sut_A.RunOneStep := FALSE;
            _sut_A.RunAllSteps := FALSE;
            _sut_A.FinishStep := TRUE;
            _sut_A.StepId := _stepId;
            _sut_N.Enabled := TRUE;
            _sut_N.RunOneStep := FALSE;
            _sut_N.RunAllSteps := FALSE;
            _sut_N.FinishStep := TRUE;
            _sut_N.StepId := _stepId;
            _sut_A.SetCurrentStep(inStepID := _currentStepId, inStepDescription := _currentStepDescription);
            _sut_N.SetCurrentStep(inStepID := _currentStepId, inStepDescription := _currentStepDescription);
            _sut_A.TcoSequencerTest := eTcoSequencerTests.NotUniqueStepId;
            _sut_N.TcoSequencerTest := eTcoSequencerTests.NotUniqueStepId;
            _sut_A.SaveNumberOfStepsInSequence();
            _sut_N.SaveNumberOfStepsInSequence();
            _plcCycleCounter := 0;
            _arranged := TRUE;
            RETURN;
        END_IF

        IF NOT _done THEN
            _sut_A.Run();
            _sut_N.Run();
            _sut_A.SaveNumberOfStepsInSequence();
            _sut_N.SaveNumberOfStepsInSequence();
            _done := _plcCycleCounter >= 2;
        END_IF

        IF _done THEN
            ProbeDoneWhen(_done);
        END_IF
        {endregion}
        {region "T516_AfterErrorRestore"}
    eTcoSequencerTests.AfterErrorRestore:
        IF NOT _arranged THEN
            _sut_A.TcoSequencerTest := eTcoSequencerTests.AfterErrorRestore;
            _sut_N.TcoSequencerTest := eTcoSequencerTests.AfterErrorRestore;
            _sut_A.SaveNumberOfStepsInSequence();
            _sut_N.SaveNumberOfStepsInSequence();
            _plcCycleCounter := 0;
            _arranged := TRUE;
            RETURN;
        END_IF

        IF NOT _done THEN
            _sut_A.Run();
            _sut_N.Run();
            _sut_A.SaveNumberOfStepsInSequence();
            _sut_N.SaveNumberOfStepsInSequence();
            _done := _plcCycleCounter >= 3;
        END_IF

        IF _done THEN
            ProbeDoneWhen(_done);
        END_IF
        {endregion}
        {region "T520_ChangeStepIdDuringExecution"}
    eTcoSequencerTests.ChangeStepIdDuringExecution:
        IF NOT _arranged THEN
            _sut_A.TcoSequencerTest := eTcoSequencerTests.ChangeStepIdDuringExecution;
            _sut_N.TcoSequencerTest := eTcoSequencerTests.ChangeStepIdDuringExecution;
            _sut_A.SetCyclicMode(); //Set sequencer into the cyclic mode
            _sut_N.SetCyclicMode(); //Set sequencer into the cyclic mode
            _sut_A.SetSequenceAsChecked(); //Set sequence as checked, so no StepID uniqueness is performed on next sequence execution
            _sut_N.SetSequenceAsChecked(); //Set sequence as checked, so no StepID uniqueness is performed on next sequence execution
            _sut_A.ClearNumberOfSteps(); //Clear internal step counters, so number of steps is going to be counted again on next sequence run
            _sut_N.ClearNumberOfSteps(); //Clear internal step counters, so number of steps is going to be counted again on next sequence run
            _sut_A.SetCurrentStep(inStepID := _currentStepId, inStepDescription := _currentStepDescription);
            _sut_N.SetCurrentStep(inStepID := _currentStepId, inStepDescription := _currentStepDescription);
            _sut_A.TotalStepNumber := _totalStepNumber;
            _sut_N.TotalStepNumber := _totalStepNumber;
            _sut_A.SaveNumberOfStepsInSequence();
            _sut_N.SaveNumberOfStepsInSequence();
            _plcCycleCounter := 0;
            _arranged := TRUE;
            RETURN;
        END_IF

        IF NOT _done THEN
            _sut_A.SequenceRun := _plcCycleCounter;
            _sut_N.SequenceRun := _plcCycleCounter;
            _sut_A.Run();
            _sut_N.Run();
            _sut_A.SaveNumberOfStepsInSequence();
            _sut_N.SaveNumberOfStepsInSequence();
        END_IF

        _done := _plcCycleCounter >= 3;
        ProbeDoneWhen(_done);
        {endregion}
        {region "T524_CommentOutPartOfRunningSequencer"}
    eTcoSequencerTests.CommentOutPartOfRunningSequencer:
        IF NOT _arranged THEN
            _sut_A.TcoSequencerTest := eTcoSequencerTests.CommentOutPartOfRunningSequencer;
            _sut_N.TcoSequencerTest := eTcoSequencerTests.CommentOutPartOfRunningSequencer;
            _sut_A.SetCyclicMode(); //Set sequencer into the cyclic mode
            _sut_N.SetCyclicMode(); //Set sequencer into the cyclic mode
            _sut_A.SetSequenceAsChecked(); //Set sequence as checked, so no StepID uniqueness is performed on next sequence execution
            _sut_N.SetSequenceAsChecked(); //Set sequence as checked, so no StepID uniqueness is performed on next sequence execution
            _sut_A.ClearNumberOfSteps(); //Clear internal step counters, so number of steps is going to be counted again on next sequence run
            _sut_N.ClearNumberOfSteps(); //Clear internal step counters, so number of steps is going to be counted again on next sequence run
            _sut_A.SetCurrentStep(inStepID := _currentStepId, inStepDescription := _currentStepDescription);
            _sut_N.SetCurrentStep(inStepID := _currentStepId, inStepDescription := _currentStepDescription);
            _sut_A.TotalStepNumber := _totalStepNumber;
            _sut_N.TotalStepNumber := _totalStepNumber;
            _sut_A.SaveNumberOfStepsInSequence();
            _sut_N.SaveNumberOfStepsInSequence();
            _plcCycleCounter := 0;
            _arranged := TRUE;
            RETURN;
        END_IF

        IF NOT _done THEN
            IF _plcCycleCounter = 3 THEN
                _sut_A.Restore();
                _sut_N.Restore();
                _sut_A.SetSequenceAsChecked(); //Set sequence as checked, so no StepID uniqueness is performed on next sequence execution
                _sut_N.SetSequenceAsChecked(); //Set sequence as checked, so no StepID uniqueness is performed on next sequence execution
                _sut_A.ClearNumberOfSteps(); //Clear internal step counters, so number of steps is going to be counted again on next sequence run
                _sut_N.ClearNumberOfSteps(); //Clear internal step counters, so number of steps is going to be counted again on next sequence run
            END_IF

            _sut_A.SequenceRun := _plcCycleCounter;
            _sut_N.SequenceRun := _plcCycleCounter;
            _sut_A.Run();
            _sut_N.Run();
            _sut_A.SaveNumberOfStepsInSequence();
            _sut_N.SaveNumberOfStepsInSequence();
        END_IF

        _done := _plcCycleCounter >= 3;
        ProbeDoneWhen(_done);
        {endregion}
        {region "T526_UncommentPartOfRunningSequencer"}
    eTcoSequencerTests.UncommentPartOfRunningSequencer:
        IF NOT _arranged THEN
            _sut_A.TcoSequencerTest := eTcoSequencerTests.UncommentPartOfRunningSequencer;
            _sut_N.TcoSequencerTest := eTcoSequencerTests.UncommentPartOfRunningSequencer;
            _sut_A.SetCyclicMode(); //Set sequencer into the cyclic mode
            _sut_N.SetCyclicMode(); //Set sequencer into the cyclic mode
            _sut_A.SetSequenceAsChecked(); //Set sequence as checked, so no StepID uniqueness is performed on next sequence execution
            _sut_N.SetSequenceAsChecked(); //Set sequence as checked, so no StepID uniqueness is performed on next sequence execution
            _sut_A.ClearNumberOfSteps(); //Clear internal step counters, so number of steps is going to be counted again on next sequence run
            _sut_N.ClearNumberOfSteps(); //Clear internal step counters, so number of steps is going to be counted again on next sequence run
            _sut_A.SetCurrentStep(inStepID := _currentStepId, inStepDescription := _currentStepDescription);
            _sut_N.SetCurrentStep(inStepID := _currentStepId, inStepDescription := _currentStepDescription);
            _sut_A.TotalStepNumber := _totalStepNumber;
            _sut_N.TotalStepNumber := _totalStepNumber;
            _sut_A.SaveNumberOfStepsInSequence();
            _sut_N.SaveNumberOfStepsInSequence();
            _plcCycleCounter := 0;
            _arranged := TRUE;
            RETURN;
        END_IF

        IF NOT _done THEN
            _sut_A.SequenceRun := _plcCycleCounter;
            _sut_N.SequenceRun := _plcCycleCounter;
            _sut_A.Run();
            _sut_N.Run();
            _sut_A.SaveNumberOfStepsInSequence();
            _sut_N.SaveNumberOfStepsInSequence();
        END_IF

        _done := _plcCycleCounter >= 2;
        ProbeDoneWhen(_done);
        {endregion}
        {region "T530_OpenCloseSequence"}
    eTcoSequencerTests.OpenCloseSequence:
        IF NOT _arranged THEN
            _sut_A.TcoSequencerTest := eTcoSequencerTests.OpenCloseSequence;
            _sut_N.TcoSequencerTest := eTcoSequencerTests.OpenCloseSequence;
            _sut_A.SetCyclicMode(); //Set sequencer into the cyclic mode
            _sut_N.SetCyclicMode(); //Set sequencer into the cyclic mode
            _sut_A.SetSequenceAsChecked(); //Set sequence as checked, so no StepID uniqueness is performed on next sequence execution
            _sut_N.SetSequenceAsChecked(); //Set sequence as checked, so no StepID uniqueness is performed on next sequence execution
            _sut_A.ClearNumberOfSteps(); //Clear internal step counters, so number of steps is going to be counted again on next sequence run
            _sut_N.ClearNumberOfSteps(); //Clear internal step counters, so number of steps is going to be counted again on next sequence run
            _sut_A.TotalStepNumber := _totalStepNumber;
            _sut_N.TotalStepNumber := _totalStepNumber;
            _sut_A.SaveNumberOfStepsInSequence();
            _sut_N.SaveNumberOfStepsInSequence();
            _plcCycleCounter := 0;
            _arranged := TRUE;
            RETURN;
        END_IF

        IF NOT _done THEN
            IF _plcCycleCounter = 1 THEN
                _sut_A.SequencerOpen();
                _sut_N.SequencerOpen();

                IF _sut_A._Step(0, TRUE, 'Step 0') THEN
                    _sut_A._StepCompleteWhen(TRUE);
                END_IF

                IF _sut_N._Step(0, TRUE, 'Step 0') THEN
                    _sut_N._StepCompleteWhen(TRUE);
                END_IF
            END_IF

            IF _plcCycleCounter = 2 THEN
                FOR i := 1 TO _totalStepNumber DO
                    _sut_A._Step(i, TRUE, CONCAT('Step ', INT_TO_STRING(i)));
                    _sut_N._Step(i, TRUE, CONCAT('Step ', INT_TO_STRING(i)));
                END_FOR

                _sut_A.SequencerClose();
                _sut_N.SequencerClose();
            END_IF

            IF _plcCycleCounter = 3 THEN
                _sut_A.SequencerOpen();
                _sut_N.SequencerOpen();
            END_IF

            IF _plcCycleCounter = 4 THEN
                IF _sut_A._Step(0, TRUE, 'Step 0') THEN
                    _sut_A._StepCompleteWhen(TRUE);
                END_IF

                IF _sut_N._Step(0, TRUE, 'Step 0') THEN
                    _sut_N._StepCompleteWhen(TRUE);
                END_IF
            END_IF

            IF _plcCycleCounter = 5 THEN
                FOR i := 1 TO _totalStepNumber DO
                    IF _sut_A._Step(i, TRUE, CONCAT('Step ', INT_TO_STRING(i))) THEN
                        _sut_A._StepCompleteWhen(TRUE);
                    END_IF

                    IF _sut_N._Step(i, TRUE, CONCAT('Step ', INT_TO_STRING(i))) THEN
                        _sut_N._StepCompleteWhen(TRUE);
                    END_IF
                END_FOR
            END_IF

            IF _plcCycleCounter = 6 THEN
                _sut_A._SequenceComplete();
                _sut_N._SequenceComplete();
                _sut_A.SequencerClose();
                _sut_N.SequencerClose();
            END_IF

            IF _plcCycleCounter = 7 THEN
                _sut_A.SequencerOpen();
                _sut_N.SequencerOpen();
            END_IF

            IF _plcCycleCounter = 8 THEN
                _sut_A.SequencerClose();
                _sut_N.SequencerClose();
            END_IF

            IF _plcCycleCounter = 9 THEN
                _sut_A.SequencerOpen();
                _sut_N.SequencerOpen();
                _sut_A._Step(0, TRUE, 'Step 0');
                _sut_N._Step(0, TRUE, 'Step 0');
                _sut_A.SequencerClose();
                _sut_N.SequencerClose();
            END_IF
        END_IF

        _done := _plcCycleCounter >= 9;
        ProbeDoneWhen(_done);
        {endregion}
        {region "T541_RequestStepFromLowerToHigher"}
    eTcoSequencerTests.RequestStepFromLowerToHigher:
        IF NOT _arranged THEN
            _sut_A.TcoSequencerTest := eTcoSequencerTests.RequestStepFromLowerToHigher;
            _sut_N.TcoSequencerTest := eTcoSequencerTests.RequestStepFromLowerToHigher;
            _sut_A.SetCyclicMode(); //Set sequencer into the cyclic mode
            _sut_N.SetCyclicMode(); //Set sequencer into the cyclic mode
            _sut_A.SetSequenceAsChecked(); //Set sequence as checked, so no StepID uniqueness is performed on next sequence execution
            _sut_N.SetSequenceAsChecked(); //Set sequence as checked, so no StepID uniqueness is performed on next sequence execution
            _sut_A.ClearNumberOfSteps(); //Clear internal step counters, so number of steps is going to be counted again on next sequence run
            _sut_N.ClearNumberOfSteps(); //Clear internal step counters, so number of steps is going to be counted again on next sequence run
            _sut_A.SetCurrentStep(inStepID := _currentStepId, inStepDescription := _currentStepDescription);
            _sut_N.SetCurrentStep(inStepID := _currentStepId, inStepDescription := _currentStepDescription);
            _sut_A.TotalStepNumber := _totalStepNumber;
            _sut_N.TotalStepNumber := _totalStepNumber;
            _sut_A.ReqStep := _reqStep;
            _sut_N.ReqStep := _reqStep;
            _sut_A.ReqStepNotExists := _reqStepNotExists;
            _sut_N.ReqStepNotExists := _reqStepNotExists;
            _sut_A.SaveNumberOfStepsInSequence();
            _sut_N.SaveNumberOfStepsInSequence();
            _plcCycleCounter := 0;
            _arranged := TRUE;
            RETURN;
        END_IF

        IF NOT _done THEN
            _sut_A.SequenceRun := _plcCycleCounter;
            _sut_N.SequenceRun := _plcCycleCounter;
            _sut_A.Run();
            _sut_N.Run();
            _sut_A.SaveNumberOfStepsInSequence();
            _sut_N.SaveNumberOfStepsInSequence();
        END_IF

        _done := _plcCycleCounter >= 2;
        ProbeDoneWhen(_done);
        {endregion}
        {region "T542_RequestStepFromHigherToLower"}
    eTcoSequencerTests.RequestStepFromHigherToLower:
        IF NOT _arranged THEN
            _sut_A.TcoSequencerTest := eTcoSequencerTests.RequestStepFromHigherToLower;
            _sut_N.TcoSequencerTest := eTcoSequencerTests.RequestStepFromHigherToLower;
            _sut_A.SetCyclicMode(); //Set sequencer into the cyclic mode
            _sut_N.SetCyclicMode(); //Set sequencer into the cyclic mode
            _sut_A.SetSequenceAsChecked(); //Set sequence as checked, so no StepID uniqueness is performed on next sequence execution
            _sut_N.SetSequenceAsChecked(); //Set sequence as checked, so no StepID uniqueness is performed on next sequence execution
            _sut_A.SetNumberOfSteps(_totalStepNumber);
            _sut_N.SetNumberOfSteps(_totalStepNumber);
            _sut_A.SetCurrentStep(inStepID := _currentStepId, inStepDescription := _currentStepDescription);
            _sut_N.SetCurrentStep(inStepID := _currentStepId, inStepDescription := _currentStepDescription);
            _sut_A.TotalStepNumber := _totalStepNumber;
            _sut_N.TotalStepNumber := _totalStepNumber;
            _sut_A.ReqStep := _reqStep;
            _sut_N.ReqStep := _reqStep;
            _sut_A.ReqStepNotExists := _reqStepNotExists;
            _sut_N.ReqStepNotExists := _reqStepNotExists;
            _sut_A.SaveNumberOfStepsInSequence();
            _sut_N.SaveNumberOfStepsInSequence();
            _plcCycleCounter := 0;
            _arranged := TRUE;
            RETURN;
        END_IF

        IF NOT _done THEN
            _sut_A.SequenceRun := _plcCycleCounter;
            _sut_N.SequenceRun := _plcCycleCounter;
            _sut_A.Run();
            _sut_N.Run();
            _sut_A.SaveNumberOfStepsInSequence();
            _sut_N.SaveNumberOfStepsInSequence();
        END_IF

        _done := _plcCycleCounter >= 2;
        ProbeDoneWhen(_done);
        {endregion}
        {region "T544_RequestStepToNotExistingStep"}
    eTcoSequencerTests.RequestStepToNotExistingStep:
        IF NOT _arranged THEN
            _sut_A.TcoSequencerTest := eTcoSequencerTests.RequestStepToNotExistingStep;
            _sut_N.TcoSequencerTest := eTcoSequencerTests.RequestStepToNotExistingStep;
            _sut_A.SetCyclicMode(); //Set sequencer into the cyclic mode
            _sut_N.SetCyclicMode(); //Set sequencer into the cyclic mode
            _sut_A.SetSequenceAsChecked(); //Set sequence as checked, so no StepID uniqueness is performed on next sequence execution
            _sut_N.SetSequenceAsChecked(); //Set sequence as checked, so no StepID uniqueness is performed on next sequence execution
            _sut_A.SetNumberOfSteps(_totalStepNumber);
            _sut_N.SetNumberOfSteps(_totalStepNumber);
            _sut_A.SetCurrentStep(inStepID := _currentStepId, inStepDescription := _currentStepDescription);
            _sut_N.SetCurrentStep(inStepID := _currentStepId, inStepDescription := _currentStepDescription);
            _sut_A.TotalStepNumber := _totalStepNumber;
            _sut_N.TotalStepNumber := _totalStepNumber;
            _sut_A.ReqStep := _reqStep;
            _sut_N.ReqStep := _reqStep;
            _sut_A.ReqStepNotExists := _reqStepNotExists;
            _sut_N.ReqStepNotExists := _reqStepNotExists;
            _sut_A.SaveNumberOfStepsInSequence();
            _sut_N.SaveNumberOfStepsInSequence();
            _plcCycleCounter := 0;
            _arranged := TRUE;
            RETURN;
        END_IF

        IF _plcCycleCounter = 4 THEN
            _sut_A.Restore();
            _sut_N.Restore();
            _sut_A.SetCyclicMode(); //Set sequencer into the cyclic mode
            _sut_N.SetCyclicMode(); //Set sequencer into the cyclic mode
            _sut_A.SetSequenceAsChecked(); //Set sequence as checked, so no StepID uniqueness is performed on next sequence execution
            _sut_N.SetSequenceAsChecked(); //Set sequence as checked, so no StepID uniqueness is performed on next sequence execution
            _sut_A.SetNumberOfSteps(_totalStepNumber);
            _sut_N.SetNumberOfSteps(_totalStepNumber);
            _sut_A.SetCurrentStep(inStepID := _currentStepId, inStepDescription := _currentStepDescription);
            _sut_N.SetCurrentStep(inStepID := _currentStepId, inStepDescription := _currentStepDescription);
            _sut_A.TotalStepNumber := _totalStepNumber;
            _sut_N.TotalStepNumber := _totalStepNumber;
        END_IF

        IF NOT _done THEN
            _sut_A.SequenceRun := _plcCycleCounter;
            _sut_N.SequenceRun := _plcCycleCounter;
            _sut_A.Run();
            _sut_N.Run();
            _sut_A.SaveNumberOfStepsInSequence();
            _sut_N.SaveNumberOfStepsInSequence();
        END_IF

        _done := _plcCycleCounter >= 4;
        ProbeDoneWhen(_done);
        {endregion}
        {region "T547_RequestStepWhilePreviousRequestStepHasNotBeenYetProcessed"}
    eTcoSequencerTests.RequestStepWhilePreviousRequestStepHasNotBeenYetProcessed:
        IF NOT _arranged THEN
            _sut_A.TcoSequencerTest := eTcoSequencerTests.RequestStepWhilePreviousRequestStepHasNotBeenYetProcessed;
            _sut_N.TcoSequencerTest := eTcoSequencerTests.RequestStepWhilePreviousRequestStepHasNotBeenYetProcessed;
            _sut_A.SetCyclicMode(); //Set sequencer into the cyclic mode
            _sut_N.SetCyclicMode(); //Set sequencer into the cyclic mode
            _sut_A.SetSequenceAsChecked(); //Set sequence as checked, so no StepID uniqueness is performed on next sequence execution
            _sut_N.SetSequenceAsChecked(); //Set sequence as checked, so no StepID uniqueness is performed on next sequence execution
            _sut_A.SetNumberOfSteps(_totalStepNumber);
            _sut_N.SetNumberOfSteps(_totalStepNumber);
            _sut_A.SetCurrentStep(inStepID := _currentStepId, inStepDescription := _currentStepDescription);
            _sut_N.SetCurrentStep(inStepID := _currentStepId, inStepDescription := _currentStepDescription);
            _sut_A.TotalStepNumber := _totalStepNumber;
            _sut_N.TotalStepNumber := _totalStepNumber;
            _sut_A.ReqStep := _reqStep;
            _sut_N.ReqStep := _reqStep;
            _sut_A.ReqStepNotExists := _reqStepNotExists;
            _sut_N.ReqStepNotExists := _reqStepNotExists;
            _sut_A.SaveNumberOfStepsInSequence();
            _sut_N.SaveNumberOfStepsInSequence();
            _plcCycleCounter := 0;
            _arranged := TRUE;
            RETURN;
        END_IF

        IF NOT _done THEN
            _sut_A.SequenceRun := _plcCycleCounter;
            _sut_N.SequenceRun := _plcCycleCounter;
            _sut_A.Run();
            _sut_N.Run();
            _sut_A.SaveNumberOfStepsInSequence();
            _sut_N.SaveNumberOfStepsInSequence();
        END_IF

        _done := TRUE;
        ProbeDoneWhen(_done);
        {endregion}
        {region "T551_DisableStepEnabledAndActiveInPreviousPLCcycle"}
    eTcoSequencerTests.DisableStepEnabledAndActiveInPreviousPLCcycle:
        IF NOT _arranged THEN
            _sut_A.TcoSequencerTest := eTcoSequencerTests.DisableStepEnabledAndActiveInPreviousPLCcycle;
            _sut_N.TcoSequencerTest := eTcoSequencerTests.DisableStepEnabledAndActiveInPreviousPLCcycle;
            _sut_A.SetCyclicMode(); //Set sequencer into the cyclic mode
            _sut_N.SetCyclicMode(); //Set sequencer into the cyclic mode
            _sut_A.SetSequenceAsChecked(); //Set sequence as checked, so no StepID uniqueness is performed on next sequence execution
            _sut_N.SetSequenceAsChecked(); //Set sequence as checked, so no StepID uniqueness is performed on next sequence execution
            _sut_A.SetNumberOfSteps(_totalStepNumber);
            _sut_N.SetNumberOfSteps(_totalStepNumber);
            _sut_A.TotalStepNumber := _totalStepNumber;
            _sut_N.TotalStepNumber := _totalStepNumber;
            _sut_A.SaveNumberOfStepsInSequence();
            _sut_N.SaveNumberOfStepsInSequence();
            _plcCycleCounter := 0;
            _arranged := TRUE;
            RETURN;
        END_IF

        IF NOT _done THEN
            IF _plcCycleCounter = 1 THEN
                _sut_A.SequencerOpen();

                IF _sut_A._Step(0, TRUE, 'Step 0') THEN
                    _sut_A._StepCompleteWhen(TRUE);
                END_IF

                FOR i := 1 TO _totalStepNumber - 2 DO
                    _sut_A._Step(i, TRUE, CONCAT('Step ', INT_TO_STRING(i)));
                END_FOR

